KUKA KRL program: EPS_2_251806_MH07A_A_20260223023033.src

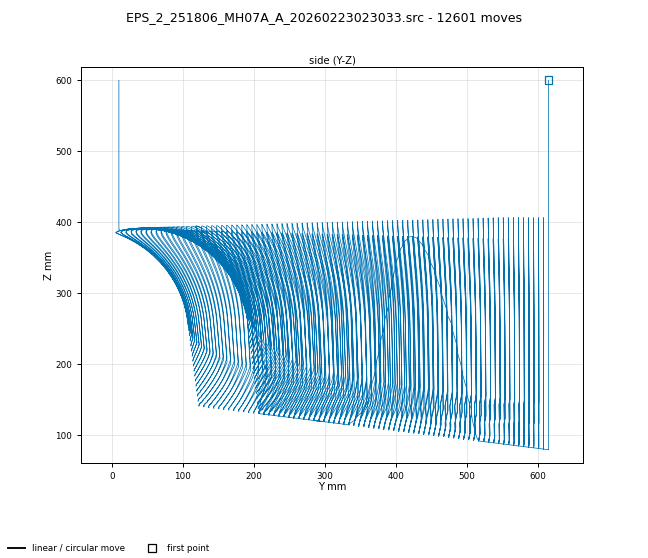
[picture p0: tool path of EPS_2_251806_MH07A_A_20260223023033.src, 12601 of 12603 moves have a stored position in this frame; points joined in program order, loops and branches not executed]
&ACCESS RVP
&REL 4
&COMMENT QRS 19112012
&PARAM EDITMASK = *
DEF PART()
EXT BAS (BAS_COMMAND :IN,REAL :IN )
INT I
BAS (#INITMOV,0 )

;KUKA QRS Post kuka4.cps  Date:22-06-2017 !

File_ID=3075

QRS_PRE_INIT()

;Init var - Until changes are made in qrs_pre_init
Outlet_Square_prg=0
Inlet_1_Square_prg=0
Inlet_2_Square_prg=0
Inlet_3_Square_prg=0
Inlet_4_Square_prg=0
Inlet_5_Square_prg=0

Outlet_1={X 0.000, Y 543.810, Z 281.000, B 0.000, E1 0.000 }
Inlet_1={X 0.000, Y 545.970, Z 251.000, B 0.000, E1 164.000 }
Outlet_1_type=251
Inlet_1_type=251
;QRS#1=Sidecore dimensions
;QRS#2=250-10" PVC SDR 35
;QRS#3=250-10" PVC SDR 35
;QRS#4=
;QRS#5=
;QRS#6=
;QRS#7=
;QRS#8=
;QRS#9=14M PSX
;QRS#10=14M PSX
;QRS#11=
;QRS#12=
;QRS#13=
;QRS#14=
;QRS#15=
;QRS#16=1220x127x686 2,25'
;QRS#17=EPS Height
;QRS#18=406,5
;QRS#19=*
;QRS#20= UPDATED VERSION 22-06-2017
;QRS#21=*
Outlet_Square=0100
Inlet_1_Square=0100
Inlet_2_Square=0
Inlet_3_Square=0
Inlet_4_Square=0
Inlet_5_Square=0
Mill_Square=1
Outlet_Square_Prg=205
Inlet_1_Square_prg=205

QRS_INIT()

$ADVANCE=5

; T1
PTP {E1 173.638,E2 173.638}
PTP {X 0,Y 615.462,A -85,B 0,C 180,E1 173.638,E2 173.638,E3 0,E4 0,E5 0,E6 0}
QRS_SPEED_INIT()
LIN {X 0,Y 615.462,Z 600,A -85,B 0,C 180,E1 173.638,E2 173.638,E3 0,E4 0,E5 0,E6 0} C_VEL
LIN {X 0,Y 615.462,Z 89.499,A -85,B 0,C 180,E1 173.638,E2 173.638} C_VEL
LIN {X 0,Y 615.462,Z 81.318,A -85,B 0,C 180,E1 173.638,E2 173.638} C_VEL
LIN {X 0,Y 615.456,Z 79.318,A -85,B 0,C 180,E1 173.452,E2 173.452} C_VEL
LIN {X 0,Y 615.494,Z 79.31,A -85,B 0,C 180,E1 170.804,E2 170.804} C_VEL
LIN {X 0,Y 615.478,Z 79.324,A -85,B 0,C 180,E1 168.142,E2 168.142} C_VEL
LIN {X 0,Y 615.453,Z 79.316,A -85,B 0,C 180,E1 165.453,E2 165.453} C_VEL
LIN {X 0,Y 615.495,Z 79.319,A -85,B 0,C 180,E1 162.733,E2 162.733} C_VEL
LIN {X 0,Y 615.448,Z 79.32,A -85,B 0,C 180,E1 159.969,E2 159.969} C_VEL
LIN {X 0,Y 615.45,Z 79.317,A -85,B 0,C 180,E1 157.664,E2 157.664} C_VEL
LIN {X 0,Y 615.497,Z 79.319,A -85,B 0,C 180,E1 155.012,E2 155.012} C_VEL
LIN {X 0,Y 615.485,Z 79.326,A -85,B 0,C 180,E1 152.826,E2 152.826} C_VEL
LIN {X 0,Y 615.437,Z 79.321,A -85,B 0,C 180,E1 150.215,E2 150.215} C_VEL
LIN {X 0,Y 615.461,Z 79.318,A -85,B 0,C 180,E1 147.674,E2 147.674} C_VEL
LIN {X 0,Y 615.498,Z 79.325,A -85,B 0,C 180,E1 145.19,E2 145.19} C_VEL
LIN {X 0,Y 615.444,Z 79.323,A -85,B 0,C 180,E1 142.759,E2 142.759} C_VEL
LIN {X 0,Y 615.46,Z 79.319,A -85,B 0,C 180,E1 139.915,E2 139.915} C_VEL
LIN {X 0,Y 615.5,Z 79.319,A -85,B 0,C 180,E1 137.653,E2 137.653} C_VEL
LIN {X 0,Y 615.431,Z 79.323,A -85,B 0,C 180,E1 134.931,E2 134.931} C_VEL
LIN {X 0,Y 615.465,Z 79.321,A -85,B 0,C 180,E1 132.083,E2 132.083} C_VEL
LIN {X 0,Y 615.489,Z 79.326,A -85,B 0,C 180,E1 129.751,E2 129.751} C_VEL
LIN {X 0,Y 615.429,Z 79.324,A -85,B 0,C 180,E1 127.247,E2 127.247} C_VEL
LIN {X 0,Y 615.431,Z 79.462,A -85,B 0,C 180,E1 126.587,E2 126.587} C_VEL
LIN {X 0,Y 615.47,Z 98.899,A -85,B 0,C 180,E1 123.78,E2 123.78} C_VEL
LIN {X 0,Y 615.473,Z 114.632,A -85,B 0,C 180,E1 121.538,E2 121.538} C_VEL
LIN {X 0,Y 615.488,Z 251.915,A -85,B 0,C 180,E1 119.892,E2 119.892} C_VEL
LIN {X 0,Y 615.49,Z 265.372,A -85,B 0,C 180,E1 119.604,E2 119.604} C_VEL
LIN {X 0,Y 615.481,Z 279.244,A -85,B 0,C 180,E1 119.173,E2 119.173} C_VEL
LIN {X 0,Y 615.488,Z 292.745,A -85,B 0,C 180,E1 118.609,E2 118.609} C_VEL
LIN {X 0,Y 615.495,Z 305.732,A -85,B 0,C 180,E1 117.916,E2 117.916} C_VEL
LIN {X 0,Y 615.497,Z 316.928,A -85,B 0,C 180,E1 117.178,E2 117.178} C_VEL
LIN {X 0,Y 615.497,Z 328.369,A -85,B 0,C 180,E1 116.262,E2 116.262} C_VEL
LIN {X 0,Y 615.494,Z 338.407,A -85,B 0,C 180,E1 115.286,E2 115.286} C_VEL
LIN {X 0,Y 615.497,Z 347.013,A -85,B 0,C 180,E1 114.272,E2 114.272} C_VEL
LIN {X 0,Y 615.496,Z 354.545,A -85,B 0,C 180,E1 113.2,E2 113.2} C_VEL
LIN {X 0,Y 615.498,Z 360.676,A -85,B 0,C 180,E1 112.137,E2 112.137} C_VEL
LIN {X 0,Y 615.498,Z 365.573,A -85,B 0,C 180,E1 111.081,E2 111.081} C_VEL
LIN {X 0,Y 615.489,Z 370.526,A -85,B 0,C 180,E1 109.686,E2 109.686} C_VEL
LIN {X 0,Y 615.497,Z 373.149,A -85,B 0,C 180,E1 108.62,E2 108.62} C_VEL
LIN {X 0,Y 615.493,Z 375.219,A -85,B 0,C 180,E1 107.271,E2 107.271} C_VEL
LIN {X 0,Y 615.493,Z 375.883,A -85,B 0,C 180,E1 105.906,E2 105.906} C_VEL
LIN {X 0,Y 615.497,Z 375.112,A -85,B 0,C 180,E1 104.55,E2 104.55} C_VEL
LIN {X 0,Y 615.495,Z 372.958,A -85,B 0,C 180,E1 103.202,E2 103.202} C_VEL
LIN {X 0,Y 615.49,Z 369.374,A -85,B 0,C 180,E1 101.862,E2 101.862} C_VEL
LIN {X 0,Y 615.495,Z 364.281,A -85,B 0,C 180,E1 100.528,E2 100.528} C_VEL
LIN {X 0,Y 615.495,Z 359.354,A -85,B 0,C 180,E1 99.531,E2 99.531} C_VEL
LIN {X 0,Y 615.495,Z 352.301,A -85,B 0,C 180,E1 98.372,E2 98.372} C_VEL
LIN {X 0,Y 615.495,Z 343.605,A -85,B 0,C 180,E1 97.216,E2 97.216} C_VEL
LIN {X 0,Y 615.497,Z 334.553,A -85,B 0,C 180,E1 96.228,E2 96.228} C_VEL
LIN {X 0,Y 615.497,Z 325.562,A -85,B 0,C 180,E1 95.406,E2 95.406} C_VEL
LIN {X 0,Y 615.498,Z 314.887,A -85,B 0,C 180,E1 94.585,E2 94.585} C_VEL
LIN {X 0,Y 615.485,Z 303.261,A -85,B 0,C 180,E1 93.847,E2 93.847} C_VEL
LIN {X 0,Y 615.495,Z 290.463,A -85,B 0,C 180,E1 93.192,E2 93.192} C_VEL
LIN {X 0,Y 615.496,Z 277.102,A -85,B 0,C 180,E1 92.66,E2 92.66} C_VEL
LIN {X 0,Y 615.47,Z 263.184,A -85,B 0,C 180,E1 92.25,E2 92.25} C_VEL
LIN {X 0,Y 615.451,Z 249.843,A -85,B 0,C 180,E1 91.985,E2 91.985} C_VEL
LIN {X 0,Y 615.447,Z 114.619,A -85,B 0,C 180,E1 90.369,E2 90.369} C_VEL
LIN {X 0,Y 615.485,Z 95.966,A -85,B 0,C 180,E1 87.71,E2 87.71} C_VEL
LIN {X 0,Y 615.485,Z 79.31,A -85,B 0,C 180,E1 85.293,E2 85.293} C_VEL
LIN {X 0,Y 615.473,Z 79.313,A -85,B 0,C 180,E1 82.785,E2 82.785} C_VEL
LIN {X 0,Y 615.499,Z 79.325,A -85,B 0,C 180,E1 80.139,E2 80.139} C_VEL
LIN {X 0,Y 615.491,Z 79.308,A -85,B 0,C 180,E1 77.471,E2 77.471} C_VEL
LIN {X 0,Y 615.472,Z 79.317,A -85,B 0,C 180,E1 74.775,E2 74.775} C_VEL
LIN {X 0,Y 615.483,Z 79.317,A -85,B 0,C 180,E1 72.044,E2 72.044} C_VEL
LIN {X 0,Y 615.479,Z 79.311,A -85,B 0,C 180,E1 69.27,E2 69.27} C_VEL
LIN {X 0,Y 615.486,Z 79.323,A -85,B 0,C 180,E1 66.445,E2 66.445} C_VEL
LIN {X 0,Y 615.485,Z 79.309,A -85,B 0,C 180,E1 63.557,E2 63.557} C_VEL
LIN {X 0,Y 615.476,Z 79.314,A -85,B 0,C 180,E1 61.343,E2 61.343} C_VEL
LIN {X 0,Y 615.488,Z 79.324,A -85,B 0,C 180,E1 58.906,E2 58.906} C_VEL
LIN {X 0,Y 615.496,Z 79.306,A -85,B 0,C 180,E1 55.98,E2 55.98} C_VEL
LIN {X 0,Y 615.49,Z 79.325,A -85,B 0,C 180,E1 53.057,E2 53.057} C_VEL
LIN {X 0,Y 615.487,Z 79.309,A -85,B 0,C 180,E1 50.251,E2 50.251} C_VEL
LIN {X 0,Y 615.478,Z 79.316,A -85,B 0,C 180,E1 47.648,E2 47.648} C_VEL
LIN {X 0,Y 615.481,Z 79.319,A -85,B 0,C 180,E1 44.933,E2 44.933} C_VEL
LIN {X 0,Y 615.481,Z 79.311,A -85,B 0,C 180,E1 42.081,E2 42.081} C_VEL
LIN {X 0,Y 615.481,Z 79.318,A -85,B 0,C 180,E1 39.746,E2 39.746} C_VEL
LIN {X 0,Y 615.477,Z 79.314,A -85,B 0,C 180,E1 36.937,E2 36.937} C_VEL
LIN {X 0,Y 615.487,Z 79.308,A -85,B 0,C 180,E1 34.703,E2 34.703} C_VEL
LIN {X 0,Y 615.481,Z 79.312,A -85,B 0,C 180,E1 32.332,E2 32.332} C_VEL
LIN {X 0,Y 615.493,Z 79.324,A -85,B 0,C 180,E1 29.798,E2 29.798} C_VEL
LIN {X 0,Y 615.476,Z 79.312,A -85,B 0,C 180,E1 27.046,E2 27.046} C_VEL
LIN {X 0,Y 615.482,Z 79.317,A -85,B 0,C 180,E1 24.269,E2 24.269} C_VEL
LIN {X 0,Y 615.475,Z 79.315,A -85,B 0,C 180,E1 21.429,E2 21.429} C_VEL
LIN {X 0,Y 615.482,Z 79.313,A -85,B 0,C 180,E1 18.607,E2 18.607} C_VEL
LIN {X 0,Y 615.481,Z 79.321,A -85,B 0,C 180,E1 15.903,E2 15.903} C_VEL
LIN {X 0,Y 615.491,Z 79.307,A -85,B 0,C 180,E1 13.198,E2 13.198} C_VEL
LIN {X 0,Y 615.488,Z 79.321,A -85,B 0,C 180,E1 10.524,E2 10.524} C_VEL
LIN {X 0,Y 615.472,Z 79.316,A -85,B 0,C 180,E1 7.873,E2 7.873} C_VEL
LIN {X 0,Y 615.492,Z 79.308,A -85,B 0,C 180,E1 5.239,E2 5.239} C_VEL
LIN {X 0,Y 615.495,Z 79.324,A -85,B 0,C 180,E1 2.616,E2 2.616} C_VEL
LIN {X 0,Y 615.472,Z 79.314,A -85,B 0,C 180,E1 -0.002,E2 -0.002} C_VEL
LIN {X 0,Y 615.489,Z 79.31,A -85,B 0,C 180,E1 -2.62,E2 -2.62} C_VEL
LIN {X 0,Y 615.49,Z 79.325,A -85,B 0,C 180,E1 -5.243,E2 -5.243} C_VEL
LIN {X 0,Y 615.47,Z 79.313,A -85,B 0,C 180,E1 -7.878,E2 -7.878} C_VEL
LIN {X 0,Y 615.486,Z 79.313,A -85,B 0,C 180,E1 -10.529,E2 -10.529} C_VEL
LIN {X 0,Y 615.475,Z 79.322,A -85,B 0,C 180,E1 -13.203,E2 -13.203} C_VEL
LIN {X 0,Y 615.486,Z 79.308,A -85,B 0,C 180,E1 -15.907,E2 -15.907} C_VEL
LIN {X 0,Y 615.487,Z 79.323,A -85,B 0,C 180,E1 -18.648,E2 -18.648} C_VEL
LIN {X 0,Y 615.469,Z 79.313,A -85,B 0,C 180,E1 -21.434,E2 -21.434} C_VEL
LIN {X 0,Y 615.487,Z 79.317,A -85,B 0,C 180,E1 -24.273,E2 -24.273} C_VEL
LIN {X 0,Y 615.466,Z 79.317,A -85,B 0,C 180,E1 -27.044,E2 -27.044} C_VEL
LIN {X 0,Y 615.492,Z 79.31,A -85,B 0,C 180,E1 -29.798,E2 -29.798} C_VEL
LIN {X 0,Y 615.489,Z 79.323,A -85,B 0,C 180,E1 -32.459,E2 -32.459} C_VEL
LIN {X 0,Y 615.464,Z 79.317,A -85,B 0,C 180,E1 -34.818,E2 -34.818} C_VEL
LIN {X 0,Y 615.48,Z 79.31,A -85,B 0,C 180,E1 -37.244,E2 -37.244} C_VEL
LIN {X 0,Y 615.496,Z 79.325,A -85,B 0,C 180,E1 -40.092,E2 -40.092} C_VEL
LIN {X 0,Y 615.473,Z 79.321,A -85,B 0,C 180,E1 -42.355,E2 -42.355} C_VEL
LIN {X 0,Y 615.476,Z 79.311,A -85,B 0,C 180,E1 -45.071,E2 -45.071} C_VEL
LIN {X 0,Y 615.494,Z 79.324,A -85,B 0,C 180,E1 -47.92,E2 -47.92} C_VEL
LIN {X 0,Y 615.465,Z 79.319,A -85,B 0,C 180,E1 -50.25,E2 -50.25} C_VEL
LIN {X 0,Y 615.49,Z 79.31,A -85,B 0,C 180,E1 -53.064,E2 -53.064} C_VEL
LIN {X 0,Y 615.469,Z 79.32,A -85,B 0,C 180,E1 -55.978,E2 -55.978} C_VEL
LIN {X 0,Y 615.461,Z 79.315,A -85,B 0,C 180,E1 -58.314,E2 -58.314} C_VEL
LIN {X 0,Y 615.476,Z 79.311,A -85,B 0,C 180,E1 -60.594,E2 -60.594} C_VEL
LIN {X 0,Y 615.478,Z 79.323,A -85,B 0,C 180,E1 -63.557,E2 -63.557} C_VEL
LIN {X 0,Y 615.459,Z 79.316,A -85,B 0,C 180,E1 -65.998,E2 -65.998} C_VEL
LIN {X 0,Y 615.485,Z 79.376,A -85,B 0,C 180,E1 -66.512,E2 -66.512} C_VEL
LIN {X 0,Y 615.489,Z 102.854,A -85,B 0,C 180,E1 -69.444,E2 -69.444} C_VEL
LIN {X 0,Y 615.492,Z 125.455,A -85,B 0,C 180,E1 -72.216,E2 -72.216} C_VEL
LIN {X 0,Y 615.493,Z 143.435,A -85,B 0,C 180,E1 -74.393,E2 -74.393} C_VEL
LIN {X 0,Y 615.477,Z 281.352,A -85,B 0,C 180,E1 -76.053,E2 -76.053} C_VEL
LIN {X 0,Y 615.489,Z 294.895,A -85,B 0,C 180,E1 -76.337,E2 -76.337} C_VEL
LIN {X 0,Y 615.488,Z 308.595,A -85,B 0,C 180,E1 -76.758,E2 -76.758} C_VEL
LIN {X 0,Y 615.494,Z 321.858,A -85,B 0,C 180,E1 -77.303,E2 -77.303} C_VEL
LIN {X 0,Y 615.483,Z 334.618,A -85,B 0,C 180,E1 -77.973,E2 -77.973} C_VEL
LIN {X 0,Y 615.499,Z 347.354,A -85,B 0,C 180,E1 -78.808,E2 -78.808} C_VEL
LIN {X 0,Y 615.498,Z 357.76,A -85,B 0,C 180,E1 -79.641,E2 -79.641} C_VEL
LIN {X 0,Y 615.496,Z 368.098,A -85,B 0,C 180,E1 -80.637,E2 -80.637} C_VEL
LIN {X 0,Y 615.497,Z 376.61,A -85,B 0,C 180,E1 -81.63,E2 -81.63} C_VEL
LIN {X 0,Y 615.496,Z 384.733,A -85,B 0,C 180,E1 -82.785,E2 -82.785} C_VEL
LIN {X 0,Y 615.497,Z 390.435,A -85,B 0,C 180,E1 -83.774,E2 -83.774} C_VEL
LIN {X 0,Y 615.495,Z 395.084,A -85,B 0,C 180,E1 -84.76,E2 -84.76} C_VEL
LIN {X 0,Y 615.496,Z 399.904,A -85,B 0,C 180,E1 -86.073,E2 -86.073} C_VEL
LIN {X 0,Y 615.495,Z 403.254,A -85,B 0,C 180,E1 -87.383,E2 -87.383} C_VEL
LIN {X 0,Y 615.49,Z 405.23,A -85,B 0,C 180,E1 -88.692,E2 -88.692} C_VEL
LIN {X 0,Y 615.493,Z 405.889,A -85,B 0,C 180,E1 -90.001,E2 -90.001} C_VEL
LIN {X 0,Y 615.49,Z 405.227,A -85,B 0,C 180,E1 -91.31,E2 -91.31} C_VEL
LIN {X 0,Y 615.495,Z 403.25,A -85,B 0,C 180,E1 -92.619,E2 -92.619} C_VEL
LIN {X 0,Y 615.496,Z 399.898,A -85,B 0,C 180,E1 -93.929,E2 -93.929} C_VEL
LIN {X 0,Y 615.495,Z 395.076,A -85,B 0,C 180,E1 -95.242,E2 -95.242} C_VEL
LIN {X 0,Y 615.495,Z 388.623,A -85,B 0,C 180,E1 -96.557,E2 -96.557} C_VEL
LIN {X 0,Y 615.498,Z 381.434,A -85,B 0,C 180,E1 -97.711,E2 -97.711} C_VEL
LIN {X 0,Y 615.497,Z 373.896,A -85,B 0,C 180,E1 -98.703,E2 -98.703} C_VEL
LIN {X 0,Y 615.496,Z 364.844,A -85,B 0,C 180,E1 -99.697,E2 -99.697} C_VEL
LIN {X 0,Y 615.497,Z 354.751,A -85,B 0,C 180,E1 -100.619,E2 -100.619} C_VEL
LIN {X 0,Y 615.498,Z 343.844,A -85,B 0,C 180,E1 -101.444,E2 -101.444} C_VEL
LIN {X 0,Y 615.484,Z 331.689,A -85,B 0,C 180,E1 -102.196,E2 -102.196} C_VEL
LIN {X 0,Y 615.486,Z 318.07,A -85,B 0,C 180,E1 -102.866,E2 -102.866} C_VEL
LIN {X 0,Y 615.488,Z 304.807,A -85,B 0,C 180,E1 -103.37,E2 -103.37} C_VEL
LIN {X 0,Y 615.487,Z 291.247,A -85,B 0,C 180,E1 -103.749,E2 -103.749} C_VEL
LIN {X 0,Y 615.478,Z 277.197,A -85,B 0,C 180,E1 -104.007,E2 -104.007} C_VEL
LIN {X 0,Y 615.493,Z 143.419,A -85,B 0,C 180,E1 -105.608,E2 -105.608} C_VEL
LIN {X 0,Y 615.483,Z 121.406,A -85,B 0,C 180,E1 -108.278,E2 -108.278} C_VEL
LIN {X 0,Y 615.475,Z 100.026,A -85,B 0,C 180,E1 -110.907,E2 -110.907} C_VEL
LIN {X 0,Y 615.483,Z 79.31,A -85,B 0,C 180,E1 -113.513,E2 -113.513} C_VEL
LIN {X 0,Y 615.466,Z 79.313,A -85,B 0,C 180,E1 -115.718,E2 -115.718} C_VEL
LIN {X 0,Y 615.49,Z 79.325,A -85,B 0,C 180,E1 -118.45,E2 -118.45} C_VEL
LIN {X 0,Y 615.487,Z 79.311,A -85,B 0,C 180,E1 -121.085,E2 -121.085} C_VEL
LIN {X 0,Y 615.468,Z 79.314,A -85,B 0,C 180,E1 -123.531,E2 -123.531} C_VEL
LIN {X 0,Y 615.471,Z 79.319,A -85,B 0,C 180,E1 -125.831,E2 -125.831} C_VEL
LIN {X 0,Y 615.492,Z 79.324,A -85,B 0,C 180,E1 -128.069,E2 -128.069} C_VEL
LIN {X 0,Y 615.482,Z 79.313,A -85,B 0,C 180,E1 -130.608,E2 -130.608} C_VEL
LIN {X 0,Y 615.471,Z 79.314,A -85,B 0,C 180,E1 -133.247,E2 -133.247} C_VEL
LIN {X 0,Y 615.49,Z 79.322,A -85,B 0,C 180,E1 -136.003,E2 -136.003} C_VEL
LIN {X 0,Y 615.481,Z 79.31,A -85,B 0,C 180,E1 -138.907,E2 -138.907} C_VEL
LIN {X 0,Y 615.475,Z 79.315,A -85,B 0,C 180,E1 -141.094,E2 -141.094} C_VEL
LIN {X 0,Y 615.484,Z 79.328,A -85,B 0,C 180,E1 -143.574,E2 -143.574} C_VEL
LIN {X 0,Y 615.494,Z 79.307,A -85,B 0,C 180,E1 -146.466,E2 -146.466} C_VEL
LIN {X 0,Y 615.484,Z 79.32,A -85,B 0,C 180,E1 -149.079,E2 -149.079} C_VEL
LIN {X 0,Y 615.477,Z 79.32,A -85,B 0,C 180,E1 -151.553,E2 -151.553} C_VEL
LIN {X 0,Y 615.486,Z 79.31,A -85,B 0,C 180,E1 -154.433,E2 -154.433} C_VEL
LIN {X 0,Y 615.484,Z 79.324,A -85,B 0,C 180,E1 -157.154,E2 -157.154} C_VEL
LIN {X 0,Y 615.484,Z 79.309,A -85,B 0,C 180,E1 -159.966,E2 -159.966} C_VEL
LIN {X 0,Y 615.491,Z 79.324,A -85,B 0,C 180,E1 -162.728,E2 -162.728} C_VEL
LIN {X 0,Y 615.471,Z 79.313,A -85,B 0,C 180,E1 -165.449,E2 -165.449} C_VEL
LIN {X 0,Y 615.486,Z 79.314,A -85,B 0,C 180,E1 -168.137,E2 -168.137} C_VEL
LIN {X 0,Y 615.475,Z 79.321,A -85,B 0,C 180,E1 -170.799,E2 -170.799} C_VEL
LIN {X 0,Y 615.478,Z 79.31,A -85,B 0,C 180,E1 -173.441,E2 -173.441} C_VEL
LIN {X 0,Y 615.491,Z 79.319,A -85,B 0,C 180,E1 -176.07,E2 -176.07} C_VEL
LIN {X 0,Y 615.462,Z 79.319,A -85,B 0,C 180,E1 -178.689,E2 -178.689} C_VEL
LIN {X 0,Y 615.484,Z 79.31,A -85,B 0,C 180,E1 -181.306,E2 -181.306} C_VEL
LIN {X 0,Y 615.49,Z 79.325,A -85,B 0,C 180,E1 -183.926,E2 -183.926} C_VEL
LIN {X 0,Y 615.456,Z 79.318,A -85,B 0,C 180,E1 -186.548,E2 -186.548} C_VEL
LIN {X 0,Y 614.803,Z 79.46,A -85,B 0,C 180,E1 -187.094,E2 -187.094} C_VEL
LIN {X 0,Y 611.99,Z 79.88,A -85,B 0,C 180,E1 -187.98,E2 -187.98} C_VEL
LIN {X 0,Y 609.6,Z 80.187,A -85,B 0,C 180,E1 -188.693,E2 -188.693} C_VEL
LIN {X 0,Y 608.559,Z 80.304,A -85,B 0,C 180,E1 -189.242,E2 -189.242} C_VEL
LIN {X 0,Y 608.466,Z 80.314,A -85,B 0,C 180,E1 -189.428,E2 -189.428} C_VEL
LIN {X 0,Y 608.45,Z 80.318,A -85,B 0,C 180,E1 -191.997,E2 -191.997} C_VEL
LIN {X 0,Y 608.427,Z 80.316,A -85,B 0,C 180,E1 -194.719,E2 -194.719} C_VEL
LIN {X 0,Y 608.449,Z 80.324,A -85,B 0,C 180,E1 -197.474,E2 -197.474} C_VEL
LIN {X 0,Y 608.432,Z 80.315,A -85,B 0,C 180,E1 -200.272,E2 -200.272} C_VEL
LIN {X 0,Y 608.454,Z 80.313,A -85,B 0,C 180,E1 -202.473,E2 -202.473} C_VEL
LIN {X 0,Y 608.44,Z 80.323,A -85,B 0,C 180,E1 -205.298,E2 -205.298} C_VEL
LIN {X 0,Y 608.43,Z 80.319,A -85,B 0,C 180,E1 -207.515,E2 -207.515} C_VEL
LIN {X 0,Y 608.425,Z 80.316,A -85,B 0,C 180,E1 -209.963,E2 -209.963} C_VEL
LIN {X 0,Y 608.438,Z 80.325,A -85,B 0,C 180,E1 -212.877,E2 -212.877} C_VEL
LIN {X 0,Y 608.417,Z 80.32,A -85,B 0,C 180,E1 -215.275,E2 -215.275} C_VEL
LIN {X 0,Y 608.434,Z 80.315,A -85,B 0,C 180,E1 -217.745,E2 -217.745} C_VEL
LIN {X 0,Y 608.437,Z 80.321,A -85,B 0,C 180,E1 -220.326,E2 -220.326} C_VEL
LIN {X 0,Y 608.413,Z 80.321,A -85,B 0,C 180,E1 -222.958,E2 -222.958} C_VEL
LIN {X 0,Y 608.406,Z 80.319,A -85,B 0,C 180,E1 -225.198,E2 -225.198} C_VEL
LIN {X 0,Y 608.443,Z 80.318,A -85,B 0,C 180,E1 -227.936,E2 -227.936} C_VEL
LIN {X 0,Y 608.408,Z 80.321,A -85,B 0,C 180,E1 -230.704,E2 -230.704} C_VEL
LIN {X 0,Y 608.433,Z 80.492,A -85,B 0,C 180,E1 -233.315,E2 -233.315} C_VEL
LIN {X 0,Y 608.523,Z 97.032,A -85,B 0,C 180,E1 -235.733,E2 -235.733} C_VEL
LIN {X 0,Y 608.499,Z 114.821,A -85,B 0,C 180,E1 -238.284,E2 -238.284} C_VEL
LIN {X 0,Y 608.618,Z 251.368,A -85,B 0,C 180,E1 -239.938,E2 -239.938} C_VEL
LIN {X 0,Y 608.587,Z 265.808,A -85,B 0,C 180,E1 -240.25,E2 -240.25} C_VEL
LIN {X 0,Y 608.552,Z 279.945,A -85,B 0,C 180,E1 -240.699,E2 -240.699} C_VEL
LIN {X 0,Y 608.556,Z 293.706,A -85,B 0,C 180,E1 -241.289,E2 -241.289} C_VEL
LIN {X 0,Y 608.537,Z 305.463,A -85,B 0,C 180,E1 -241.924,E2 -241.924} C_VEL
LIN {X 0,Y 608.524,Z 316.772,A -85,B 0,C 180,E1 -242.671,E2 -242.671} C_VEL
LIN {X 0,Y 608.494,Z 328.312,A -85,B 0,C 180,E1 -243.597,E2 -243.597} C_VEL
LIN {X 0,Y 608.47,Z 338.13,A -85,B 0,C 180,E1 -244.55,E2 -244.55} C_VEL
LIN {X 0,Y 608.472,Z 347.642,A -85,B 0,C 180,E1 -245.673,E2 -245.673} C_VEL
LIN {X 0,Y 608.452,Z 354.806,A -85,B 0,C 180,E1 -246.695,E2 -246.695} C_VEL
LIN {X 0,Y 608.452,Z 361.907,A -85,B 0,C 180,E1 -247.95,E2 -247.95} C_VEL
LIN {X 0,Y 608.442,Z 366.736,A -85,B 0,C 180,E1 -249.017,E2 -249.017} C_VEL
LIN {X 0,Y 608.43,Z 370.458,A -85,B 0,C 180,E1 -250.076,E2 -250.076} C_VEL
LIN {X 0,Y 608.423,Z 373.589,A -85,B 0,C 180,E1 -251.285,E2 -251.285} C_VEL
LIN {X 0,Y 608.414,Z 375.595,A -85,B 0,C 180,E1 -252.521,E2 -252.521} C_VEL
LIN {X 0,Y 608.429,Z 376.473,A -85,B 0,C 180,E1 -253.904,E2 -253.904} C_VEL
LIN {X 0,Y 608.42,Z 375.927,A -85,B 0,C 180,E1 -255.277,E2 -255.277} C_VEL
LIN {X 0,Y 608.436,Z 373.942,A -85,B 0,C 180,E1 -256.642,E2 -256.642} C_VEL
LIN {X 0,Y 608.432,Z 370.506,A -85,B 0,C 180,E1 -257.999,E2 -257.999} C_VEL
LIN {X 0,Y 608.434,Z 365.561,A -85,B 0,C 180,E1 -259.349,E2 -259.349} C_VEL
LIN {X 0,Y 608.463,Z 360.794,A -85,B 0,C 180,E1 -260.358,E2 -260.358} C_VEL
LIN {X 0,Y 608.458,Z 353.91,A -85,B 0,C 180,E1 -261.53,E2 -261.53} C_VEL
LIN {X 0,Y 608.463,Z 345.405,A -85,B 0,C 180,E1 -262.7,E2 -262.7} C_VEL
LIN {X 0,Y 608.48,Z 336.577,A -85,B 0,C 180,E1 -263.7,E2 -263.7} C_VEL
LIN {X 0,Y 608.497,Z 325.954,A -85,B 0,C 180,E1 -264.698,E2 -264.698} C_VEL
LIN {X 0,Y 608.516,Z 314.119,A -85,B 0,C 180,E1 -265.611,E2 -265.611} C_VEL
LIN {X 0,Y 608.528,Z 302.23,A -85,B 0,C 180,E1 -266.357,E2 -266.357} C_VEL
LIN {X 0,Y 608.548,Z 289.045,A -85,B 0,C 180,E1 -267.02,E2 -267.02} C_VEL
LIN {X 0,Y 608.578,Z 275.168,A -85,B 0,C 180,E1 -267.558,E2 -267.558} C_VEL
LIN {X 0,Y 608.584,Z 261.299,A -85,B 0,C 180,E1 -267.952,E2 -267.952} C_VEL
LIN {X 0,Y 608.564,Z 246.752,A -85,B 0,C 180,E1 -268.221,E2 -268.221} C_VEL
LIN {X 0,Y 608.487,Z 115.112,A -85,B 0,C 180,E1 -269.803,E2 -269.803} C_VEL
LIN {X 0,Y 608.452,Z 114.575,A -85,B 0,C 180,E1 -269.834,E2 -269.834} C_VEL
LIN {X 0,Y 608.542,Z 95.029,A -85,B 0,C 180,E1 -272.647,E2 -272.647} C_VEL
LIN {X 0,Y 608.457,Z 80.314,A -85,B 0,C 180,E1 -274.803,E2 -274.803} C_VEL
LIN {X 0,Y 608.462,Z 80.313,A -85,B 0,C 180,E1 -277.298,E2 -277.298} C_VEL
LIN {X 0,Y 608.463,Z 80.32,A -85,B 0,C 180,E1 -279.976,E2 -279.976} C_VEL
LIN {X 0,Y 608.473,Z 80.31,A -85,B 0,C 180,E1 -282.676,E2 -282.676} C_VEL
LIN {X 0,Y 608.458,Z 80.318,A -85,B 0,C 180,E1 -285.405,E2 -285.405} C_VEL
LIN {X 0,Y 608.442,Z 80.322,A -85,B 0,C 180,E1 -287.476,E2 -287.476} C_VEL
LIN {X 0,Y 608.458,Z 80.313,A -85,B 0,C 180,E1 -290.273,E2 -290.273} C_VEL
LIN {X 0,Y 608.462,Z 80.311,A -85,B 0,C 180,E1 -292.487,E2 -292.487} C_VEL
LIN {X 0,Y 608.445,Z 80.323,A -85,B 0,C 180,E1 -295.3,E2 -295.3} C_VEL
LIN {X 0,Y 608.442,Z 80.321,A -85,B 0,C 180,E1 -297.517,E2 -297.517} C_VEL
LIN {X 0,Y 608.485,Z 80.309,A -85,B 0,C 180,E1 -299.982,E2 -299.982} C_VEL
LIN {X 0,Y 608.448,Z 80.319,A -85,B 0,C 180,E1 -302.879,E2 -302.879} C_VEL
LIN {X 0,Y 608.464,Z 80.318,A -85,B 0,C 180,E1 -305.275,E2 -305.275} C_VEL
LIN {X 0,Y 608.464,Z 80.312,A -85,B 0,C 180,E1 -307.745,E2 -307.745} C_VEL
LIN {X 0,Y 608.448,Z 80.315,A -85,B 0,C 180,E1 -310.334,E2 -310.334} C_VEL
LIN {X 0,Y 608.447,Z 80.321,A -85,B 0,C 180,E1 -312.959,E2 -312.959} C_VEL
LIN {X 0,Y 608.455,Z 80.312,A -85,B 0,C 180,E1 -315.735,E2 -315.735} C_VEL
LIN {X 0,Y 608.458,Z 80.313,A -85,B 0,C 180,E1 -317.943,E2 -317.943} C_VEL
LIN {X 0,Y 608.461,Z 80.32,A -85,B 0,C 180,E1 -320.702,E2 -320.702} C_VEL
LIN {X 0,Y 608.448,Z 80.315,A -85,B 0,C 180,E1 -323.089,E2 -323.089} C_VEL
LIN {X 0,Y 608.466,Z 80.311,A -85,B 0,C 180,E1 -325.535,E2 -325.535} C_VEL
LIN {X 0,Y 608.461,Z 80.315,A -85,B 0,C 180,E1 -327.909,E2 -327.909} C_VEL
LIN {X 0,Y 608.476,Z 80.319,A -85,B 0,C 180,E1 -330.225,E2 -330.225} C_VEL
LIN {X 0,Y 608.465,Z 80.313,A -85,B 0,C 180,E1 -332.793,E2 -332.793} C_VEL
LIN {X 0,Y 608.448,Z 80.314,A -85,B 0,C 180,E1 -335.432,E2 -335.432} C_VEL
LIN {X 0,Y 608.461,Z 80.317,A -85,B 0,C 180,E1 -338.311,E2 -338.311} C_VEL
LIN {X 0,Y 608.445,Z 80.314,A -85,B 0,C 180,E1 -341.133,E2 -341.133} C_VEL
LIN {X 0,Y 608.456,Z 80.322,A -85,B 0,C 180,E1 -343.909,E2 -343.909} C_VEL
LIN {X 0,Y 608.464,Z 80.311,A -85,B 0,C 180,E1 -346.646,E2 -346.646} C_VEL
LIN {X 0,Y 608.464,Z 80.316,A -85,B 0,C 180,E1 -349.353,E2 -349.353} C_VEL
LIN {X 0,Y 608.466,Z 80.314,A -85,B 0,C 180,E1 -352.035,E2 -352.035} C_VEL
LIN {X 0,Y 608.469,Z 80.311,A -85,B 0,C 180,E1 -354.701,E2 -354.701} C_VEL
LIN {X 0,Y 608.484,Z 80.318,A -85,B 0,C 180,E1 -357.354,E2 -357.354} C_VEL
LIN {X 0,Y 608.463,Z 80.313,A -85,B 0,C 180,E1 -360.002,E2 -360.002} C_VEL
LIN {X 0,Y 608.479,Z 80.311,A -85,B 0,C 180,E1 -362.65,E2 -362.65} C_VEL
LIN {X 0,Y 608.467,Z 80.319,A -85,B 0,C 180,E1 -365.304,E2 -365.304} C_VEL
LIN {X 0,Y 608.465,Z 80.311,A -85,B 0,C 180,E1 -367.969,E2 -367.969} C_VEL
LIN {X 0,Y 608.465,Z 80.315,A -85,B 0,C 180,E1 -370.652,E2 -370.652} C_VEL
LIN {X 0,Y 608.454,Z 80.316,A -85,B 0,C 180,E1 -373.358,E2 -373.358} C_VEL
LIN {X 0,Y 608.46,Z 80.312,A -85,B 0,C 180,E1 -376.096,E2 -376.096} C_VEL
LIN {X 0,Y 608.45,Z 80.322,A -85,B 0,C 180,E1 -378.871,E2 -378.871} C_VEL
LIN {X 0,Y 608.46,Z 80.312,A -85,B 0,C 180,E1 -381.693,E2 -381.693} C_VEL
LIN {X 0,Y 608.447,Z 80.324,A -85,B 0,C 180,E1 -384.573,E2 -384.573} C_VEL
LIN {X 0,Y 608.462,Z 80.312,A -85,B 0,C 180,E1 -387.207,E2 -387.207} C_VEL
LIN {X 0,Y 608.47,Z 80.314,A -85,B 0,C 180,E1 -389.974,E2 -389.974} C_VEL
LIN {X 0,Y 608.452,Z 80.315,A -85,B 0,C 180,E1 -392.881,E2 -392.881} C_VEL
LIN {X 0,Y 608.439,Z 80.314,A -85,B 0,C 180,E1 -395.279,E2 -395.279} C_VEL
LIN {X 0,Y 608.47,Z 80.32,A -85,B 0,C 180,E1 -398.243,E2 -398.243} C_VEL
LIN {X 0,Y 608.462,Z 80.312,A -85,B 0,C 180,E1 -401.344,E2 -401.344} C_VEL
LIN {X 0,Y 608.452,Z 80.318,A -85,B 0,C 180,E1 -404.265,E2 -404.265} C_VEL
LIN {X 0,Y 608.444,Z 80.314,A -85,B 0,C 180,E1 -407.041,E2 -407.041} C_VEL
LIN {X 0,Y 608.454,Z 80.321,A -85,B 0,C 180,E1 -409.698,E2 -409.698} C_VEL
LIN {X 0,Y 608.46,Z 80.314,A -85,B 0,C 180,E1 -412.255,E2 -412.255} C_VEL
LIN {X 0,Y 608.453,Z 80.315,A -85,B 0,C 180,E1 -415.095,E2 -415.095} C_VEL
LIN {X 0,Y 608.46,Z 80.316,A -85,B 0,C 180,E1 -417.907,E2 -417.907} C_VEL
LIN {X 0,Y 608.446,Z 80.314,A -85,B 0,C 180,E1 -420.221,E2 -420.221} C_VEL
LIN {X 0,Y 608.481,Z 80.311,A -85,B 0,C 180,E1 -422.793,E2 -422.793} C_VEL
LIN {X 0,Y 608.445,Z 80.323,A -85,B 0,C 180,E1 -425.43,E2 -425.43} C_VEL
LIN {X 0,Y 608.477,Z 80.436,A -85,B 0,C 180,E1 -426.36,E2 -426.36} C_VEL
LIN {X 0,Y 608.596,Z 97.216,A -85,B 0,C 180,E1 -428.492,E2 -428.492} C_VEL
LIN {X 0,Y 608.532,Z 119.494,A -85,B 0,C 180,E1 -431.268,E2 -431.268} C_VEL
LIN {X 0,Y 608.521,Z 142.434,A -85,B 0,C 180,E1 -434.081,E2 -434.081} C_VEL
LIN {X 0,Y 608.514,Z 143.582,A -85,B 0,C 180,E1 -434.221,E2 -434.221} C_VEL
LIN {X 0,Y 608.598,Z 281.51,A -85,B 0,C 180,E1 -435.895,E2 -435.895} C_VEL
LIN {X 0,Y 608.603,Z 295.662,A -85,B 0,C 180,E1 -436.201,E2 -436.201} C_VEL
LIN {X 0,Y 608.579,Z 309.738,A -85,B 0,C 180,E1 -436.647,E2 -436.647} C_VEL
LIN {X 0,Y 608.554,Z 321.905,A -85,B 0,C 180,E1 -437.156,E2 -437.156} C_VEL
LIN {X 0,Y 608.511,Z 334.698,A -85,B 0,C 180,E1 -437.833,E2 -437.833} C_VEL
LIN {X 0,Y 608.499,Z 347.485,A -85,B 0,C 180,E1 -438.678,E2 -438.678} C_VEL
LIN {X 0,Y 608.495,Z 357.943,A -85,B 0,C 180,E1 -439.52,E2 -439.52} C_VEL
LIN {X 0,Y 608.479,Z 368.344,A -85,B 0,C 180,E1 -440.528,E2 -440.528} C_VEL
LIN {X 0,Y 608.464,Z 376.922,A -85,B 0,C 180,E1 -441.532,E2 -441.532} C_VEL
LIN {X 0,Y 608.461,Z 385.119,A -85,B 0,C 180,E1 -442.702,E2 -442.702} C_VEL
LIN {X 0,Y 608.444,Z 391.55,A -85,B 0,C 180,E1 -443.832,E2 -443.832} C_VEL
LIN {X 0,Y 608.435,Z 396.965,A -85,B 0,C 180,E1 -445.031,E2 -445.031} C_VEL
LIN {X 0,Y 608.434,Z 400.444,A -85,B 0,C 180,E1 -446.027,E2 -446.027} C_VEL
LIN {X 0,Y 608.423,Z 403.833,A -85,B 0,C 180,E1 -447.353,E2 -447.353} C_VEL
LIN {X 0,Y 608.442,Z 405.832,A -85,B 0,C 180,E1 -448.677,E2 -448.677} C_VEL
LIN {X 0,Y 608.433,Z 406.5,A -85,B 0,C 180,E1 -450.001,E2 -450.001} C_VEL
LIN {X 0,Y 608.442,Z 405.829,A -85,B 0,C 180,E1 -451.325,E2 -451.325} C_VEL
LIN {X 0,Y 608.423,Z 403.829,A -85,B 0,C 180,E1 -452.649,E2 -452.649} C_VEL
LIN {X 0,Y 608.434,Z 400.438,A -85,B 0,C 180,E1 -453.975,E2 -453.975} C_VEL
LIN {X 0,Y 608.439,Z 395.564,A -85,B 0,C 180,E1 -455.303,E2 -455.303} C_VEL
LIN {X 0,Y 608.447,Z 389.207,A -85,B 0,C 180,E1 -456.604,E2 -456.604} C_VEL
LIN {X 0,Y 608.454,Z 381.791,A -85,B 0,C 180,E1 -457.801,E2 -457.801} C_VEL
LIN {X 0,Y 608.473,Z 372.815,A -85,B 0,C 180,E1 -458.972,E2 -458.972} C_VEL
LIN {X 0,Y 608.473,Z 363.381,A -85,B 0,C 180,E1 -459.978,E2 -459.978} C_VEL
LIN {X 0,Y 608.506,Z 352.049,A -85,B 0,C 180,E1 -460.973,E2 -460.973} C_VEL
LIN {X 0,Y 608.531,Z 340.134,A -85,B 0,C 180,E1 -461.83,E2 -461.83} C_VEL
LIN {X 0,Y 608.53,Z 327.055,A -85,B 0,C 180,E1 -462.592,E2 -462.592} C_VEL
LIN {X 0,Y 608.55,Z 314.149,A -85,B 0,C 180,E1 -463.185,E2 -463.185} C_VEL
LIN {X 0,Y 608.59,Z 300.148,A -85,B 0,C 180,E1 -463.673,E2 -463.673} C_VEL
LIN {X 0,Y 608.602,Z 286.402,A -85,B 0,C 180,E1 -464.014,E2 -464.014} C_VEL
LIN {X 0,Y 608.591,Z 270.086,A -85,B 0,C 180,E1 -464.259,E2 -464.259} C_VEL
LIN {X 0,Y 608.53,Z 143.566,A -85,B 0,C 180,E1 -465.781,E2 -465.781} C_VEL
LIN {X 0,Y 608.537,Z 121.421,A -85,B 0,C 180,E1 -468.494,E2 -468.494} C_VEL
LIN {X 0,Y 608.561,Z 100.026,A -85,B 0,C 180,E1 -471.156,E2 -471.156} C_VEL
LIN {X 0,Y 608.57,Z 80.95,A -85,B 0,C 180,E1 -473.57,E2 -473.57} C_VEL
LIN {X 0,Y 608.447,Z 80.316,A -85,B 0,C 180,E1 -473.666,E2 -473.666} C_VEL
LIN {X 0,Y 608.434,Z 80.317,A -85,B 0,C 180,E1 -476.037,E2 -476.037} C_VEL
LIN {X 0,Y 608.477,Z 80.319,A -85,B 0,C 180,E1 -478.62,E2 -478.62} C_VEL
LIN {X 0,Y 608.449,Z 80.314,A -85,B 0,C 180,E1 -481.318,E2 -481.318} C_VEL
LIN {X 0,Y 608.454,Z 80.315,A -85,B 0,C 180,E1 -483.731,E2 -483.731} C_VEL
LIN {X 0,Y 608.45,Z 80.321,A -85,B 0,C 180,E1 -486.093,E2 -486.093} C_VEL
LIN {X 0,Y 608.477,Z 80.313,A -85,B 0,C 180,E1 -488.588,E2 -488.588} C_VEL
LIN {X 0,Y 608.453,Z 80.314,A -85,B 0,C 180,E1 -491.34,E2 -491.34} C_VEL
LIN {X 0,Y 608.458,Z 80.317,A -85,B 0,C 180,E1 -494.263,E2 -494.263} C_VEL
LIN {X 0,Y 608.449,Z 80.314,A -85,B 0,C 180,E1 -497.039,E2 -497.039} C_VEL
LIN {X 0,Y 608.464,Z 80.322,A -85,B 0,C 180,E1 -499.696,E2 -499.696} C_VEL
LIN {X 0,Y 608.468,Z 80.312,A -85,B 0,C 180,E1 -502.252,E2 -502.252} C_VEL
LIN {X 0,Y 608.447,Z 80.317,A -85,B 0,C 180,E1 -505.096,E2 -505.096} C_VEL
LIN {X 0,Y 608.464,Z 80.314,A -85,B 0,C 180,E1 -507.904,E2 -507.904} C_VEL
LIN {X 0,Y 608.474,Z 80.31,A -85,B 0,C 180,E1 -510.219,E2 -510.219} C_VEL
LIN {X 0,Y 608.478,Z 80.313,A -85,B 0,C 180,E1 -512.794,E2 -512.794} C_VEL
LIN {X 0,Y 608.45,Z 80.318,A -85,B 0,C 180,E1 -515.427,E2 -515.427} C_VEL
LIN {X 0,Y 608.466,Z 80.312,A -85,B 0,C 180,E1 -518.307,E2 -518.307} C_VEL
LIN {X 0,Y 608.467,Z 80.315,A -85,B 0,C 180,E1 -521.287,E2 -521.287} C_VEL
LIN {X 0,Y 608.459,Z 80.312,A -85,B 0,C 180,E1 -523.904,E2 -523.904} C_VEL
LIN {X 0,Y 608.466,Z 80.321,A -85,B 0,C 180,E1 -526.642,E2 -526.642} C_VEL
LIN {X 0,Y 608.452,Z 80.313,A -85,B 0,C 180,E1 -529.348,E2 -529.348} C_VEL
LIN {X 0,Y 608.478,Z 80.313,A -85,B 0,C 180,E1 -532.031,E2 -532.031} C_VEL
LIN {X 0,Y 608.451,Z 80.318,A -85,B 0,C 180,E1 -534.696,E2 -534.696} C_VEL
LIN {X 0,Y 608.473,Z 80.31,A -85,B 0,C 180,E1 -537.35,E2 -537.35} C_VEL
LIN {X 0,Y 608.484,Z 80.317,A -85,B 0,C 180,E1 -539.998,E2 -539.998} C_VEL
LIN {X 0,Y 608.455,Z 80.314,A -85,B 0,C 180,E1 -542.646,E2 -542.646} C_VEL
LIN {X 0,Y 608.468,Z 80.312,A -85,B 0,C 180,E1 -545.299,E2 -545.299} C_VEL
LIN {X 0,Y 608.474,Z 80.318,A -85,B 0,C 180,E1 -547.965,E2 -547.965} C_VEL
LIN {X 0,Y 608.466,Z 80.314,A -85,B 0,C 180,E1 -549.428,E2 -549.428} C_VEL
LIN {X 0,Y 607.779,Z 80.404,A -85,B 0,C 180,E1 -549.981,E2 -549.981} C_VEL
LIN {X 0,Y 604.92,Z 80.758,A -85,B 0,C 180,E1 -550.878,E2 -550.878} C_VEL
LIN {X 0,Y 602.516,Z 81.061,A -85,B 0,C 180,E1 -551.599,E2 -551.599} C_VEL
LIN {X 0,Y 601.482,Z 81.184,A -85,B 0,C 180,E1 -552.156,E2 -552.156} C_VEL
LIN {X 0,Y 601.397,Z 81.193,A -85,B 0,C 180,E1 -552.344,E2 -552.344} C_VEL
LIN {X 0,Y 601.4,Z 81.193,A -85,B 0,C 180,E1 -554.895,E2 -554.895} C_VEL
LIN {X 0,Y 601.408,Z 81.193,A -85,B 0,C 180,E1 -556.984,E2 -556.984} C_VEL
LIN {X 0,Y 601.39,Z 81.196,A -85,B 0,C 180,E1 -559.807,E2 -559.807} C_VEL
LIN {X 0,Y 601.407,Z 81.192,A -85,B 0,C 180,E1 -562.68,E2 -562.68} C_VEL
LIN {X 0,Y 601.39,Z 81.198,A -85,B 0,C 180,E1 -564.876,E2 -564.876} C_VEL
LIN {X 0,Y 601.407,Z 81.196,A -85,B 0,C 180,E1 -567.36,E2 -567.36} C_VEL
LIN {X 0,Y 601.391,Z 81.196,A -85,B 0,C 180,E1 -569.391,E2 -569.391} C_VEL
LIN {X 0,Y 601.38,Z 81.194,A -85,B 0,C 180,E1 -571.724,E2 -571.724} C_VEL
LIN {X 0,Y 601.403,Z 81.192,A -85,B 0,C 180,E1 -574.116,E2 -574.116} C_VEL
LIN {X 0,Y 601.386,Z 81.201,A -85,B 0,C 180,E1 -576.58,E2 -576.58} C_VEL
LIN {X 0,Y 601.375,Z 81.198,A -85,B 0,C 180,E1 -579.125,E2 -579.125} C_VEL
LIN {X 0,Y 601.395,Z 81.193,A -85,B 0,C 180,E1 -581.763,E2 -581.763} C_VEL
LIN {X 0,Y 601.404,Z 81.2,A -85,B 0,C 180,E1 -584.532,E2 -584.532} C_VEL
LIN {X 0,Y 601.352,Z 81.198,A -85,B 0,C 180,E1 -587.323,E2 -587.323} C_VEL
LIN {X 0,Y 601.378,Z 81.202,A -85,B 0,C 180,E1 -590.001,E2 -590.001} C_VEL
LIN {X 0,Y 601.402,Z 81.196,A -85,B 0,C 180,E1 -592.616,E2 -592.616} C_VEL
LIN {X 0,Y 601.38,Z 81.291,A -85,B 0,C 180,E1 -593.18,E2 -593.18} C_VEL
LIN {X 0,Y 601.532,Z 89.657,A -85,B 0,C 180,E1 -594.426,E2 -594.426} C_VEL
LIN {X 0,Y 601.493,Z 106.192,A -85,B 0,C 180,E1 -596.851,E2 -596.851} C_VEL
LIN {X 0,Y 601.473,Z 114.651,A -85,B 0,C 180,E1 -598.079,E2 -598.079} C_VEL
LIN {X 0,Y 601.815,Z 118.473,A -85,B 0,C 180,E1 -598.149,E2 -598.149} C_VEL
LIN {X 0,Y 601.735,Z 251.743,A -85,B 0,C 180,E1 -599.78,E2 -599.78} C_VEL
LIN {X 0,Y 601.693,Z 265.901,A -85,B 0,C 180,E1 -600.091,E2 -600.091} C_VEL
LIN {X 0,Y 601.647,Z 279.392,A -85,B 0,C 180,E1 -600.522,E2 -600.522} C_VEL
LIN {X 0,Y 601.598,Z 292.907,A -85,B 0,C 180,E1 -601.099,E2 -601.099} C_VEL
LIN {X 0,Y 601.573,Z 305.107,A -85,B 0,C 180,E1 -601.76,E2 -601.76} C_VEL
LIN {X 0,Y 601.524,Z 316.93,A -85,B 0,C 180,E1 -602.549,E2 -602.549} C_VEL
LIN {X 0,Y 601.456,Z 328.058,A -85,B 0,C 180,E1 -603.451,E2 -603.451} C_VEL
LIN {X 0,Y 601.417,Z 337.583,A -85,B 0,C 180,E1 -604.381,E2 -604.381} C_VEL
LIN {X 0,Y 601.415,Z 346.684,A -85,B 0,C 180,E1 -605.448,E2 -605.448} C_VEL
LIN {X 0,Y 601.393,Z 354.676,A -85,B 0,C 180,E1 -606.588,E2 -606.588} C_VEL
LIN {X 0,Y 601.365,Z 361.12,A -85,B 0,C 180,E1 -607.718,E2 -607.718} C_VEL
LIN {X 0,Y 601.374,Z 365.898,A -85,B 0,C 180,E1 -608.759,E2 -608.759} C_VEL
LIN {X 0,Y 601.332,Z 369.834,A -85,B 0,C 180,E1 -609.831,E2 -609.831} C_VEL
LIN {X 0,Y 601.334,Z 373.461,A -85,B 0,C 180,E1 -611.192,E2 -611.192} C_VEL
LIN {X 0,Y 601.307,Z 375.369,A -85,B 0,C 180,E1 -612.308,E2 -612.308} C_VEL
LIN {X 0,Y 601.343,Z 376.428,A -85,B 0,C 180,E1 -613.71,E2 -613.71} C_VEL
LIN {X 0,Y 601.311,Z 376.065,A -85,B 0,C 180,E1 -615.099,E2 -615.099} C_VEL
LIN {X 0,Y 601.361,Z 375.211,A -85,B 0,C 180,E1 -615.914,E2 -615.914} C_VEL
LIN {X 0,Y 601.325,Z 372.88,A -85,B 0,C 180,E1 -617.169,E2 -617.169} C_VEL
LIN {X 0,Y 601.348,Z 368.928,A -85,B 0,C 180,E1 -618.539,E2 -618.539} C_VEL
LIN {X 0,Y 601.347,Z 363.391,A -85,B 0,C 180,E1 -619.903,E2 -619.903} C_VEL
LIN {X 0,Y 601.383,Z 357.148,A -85,B 0,C 180,E1 -621.091,E2 -621.091} C_VEL
LIN {X 0,Y 601.382,Z 349.408,A -85,B 0,C 180,E1 -622.276,E2 -622.276} C_VEL
LIN {X 0,Y 601.44,Z 340.204,A -85,B 0,C 180,E1 -623.42,E2 -623.42} C_VEL
LIN {X 0,Y 601.455,Z 329.97,A -85,B 0,C 180,E1 -624.467,E2 -624.467} C_VEL
LIN {X 0,Y 601.497,Z 318.973,A -85,B 0,C 180,E1 -625.392,E2 -625.392} C_VEL
LIN {X 0,Y 601.532,Z 306.751,A -85,B 0,C 180,E1 -626.231,E2 -626.231} C_VEL
LIN {X 0,Y 601.588,Z 294.726,A -85,B 0,C 180,E1 -626.902,E2 -626.902} C_VEL
LIN {X 0,Y 601.638,Z 281.47,A -85,B 0,C 180,E1 -627.488,E2 -627.488} C_VEL
LIN {X 0,Y 601.683,Z 266.927,A -85,B 0,C 180,E1 -627.97,E2 -627.97} C_VEL
LIN {X 0,Y 601.682,Z 253.205,A -85,B 0,C 180,E1 -628.284,E2 -628.284} C_VEL
LIN {X 0,Y 601.713,Z 227.828,A -85,B 0,C 180,E1 -628.619,E2 -628.619} C_VEL
LIN {X 0,Y 601.749,Z 116.429,A -85,B 0,C 180,E1 -629.968,E2 -629.968} C_VEL
LIN {X 0,Y 601.438,Z 114.738,A -85,B 0,C 180,E1 -629.999,E2 -629.999} C_VEL
LIN {X 0,Y 601.556,Z 96.344,A -85,B 0,C 180,E1 -632.678,E2 -632.678} C_VEL
LIN {X 0,Y 601.501,Z 81.611,A -85,B 0,C 180,E1 -634.858,E2 -634.858} C_VEL
LIN {X 0,Y 601.43,Z 81.191,A -85,B 0,C 180,E1 -634.943,E2 -634.943} C_VEL
LIN {X 0,Y 601.428,Z 81.191,A -85,B 0,C 180,E1 -637.384,E2 -637.384} C_VEL
LIN {X 0,Y 601.436,Z 81.193,A -85,B 0,C 180,E1 -640.094,E2 -640.094} C_VEL
LIN {X 0,Y 601.441,Z 81.187,A -85,B 0,C 180,E1 -642.827,E2 -642.827} C_VEL
LIN {X 0,Y 601.411,Z 81.199,A -85,B 0,C 180,E1 -645.59,E2 -645.59} C_VEL
LIN {X 0,Y 601.39,Z 81.201,A -85,B 0,C 180,E1 -647.687,E2 -647.687} C_VEL
LIN {X 0,Y 601.421,Z 81.189,A -85,B 0,C 180,E1 -650.521,E2 -650.521} C_VEL
LIN {X 0,Y 601.409,Z 81.2,A -85,B 0,C 180,E1 -653.41,E2 -653.41} C_VEL
LIN {X 0,Y 601.395,Z 81.192,A -85,B 0,C 180,E1 -656.363,E2 -656.363} C_VEL
LIN {X 0,Y 601.424,Z 81.191,A -85,B 0,C 180,E1 -658.795,E2 -658.795} C_VEL
LIN {X 0,Y 601.416,Z 81.195,A -85,B 0,C 180,E1 -661.461,E2 -661.461} C_VEL
LIN {X 0,Y 601.415,Z 81.189,A -85,B 0,C 180,E1 -664.118,E2 -664.118} C_VEL
LIN {X 0,Y 601.4,Z 81.195,A -85,B 0,C 180,E1 -666.582,E2 -666.582} C_VEL
LIN {X 0,Y 601.429,Z 81.189,A -85,B 0,C 180,E1 -669.54,E2 -669.54} C_VEL
LIN {X 0,Y 601.415,Z 81.196,A -85,B 0,C 180,E1 -672.596,E2 -672.596} C_VEL
LIN {X 0,Y 601.426,Z 81.189,A -85,B 0,C 180,E1 -675.487,E2 -675.487} C_VEL
LIN {X 0,Y 601.414,Z 81.196,A -85,B 0,C 180,E1 -678.406,E2 -678.406} C_VEL
LIN {X 0,Y 601.42,Z 81.194,A -85,B 0,C 180,E1 -680.879,E2 -680.879} C_VEL
LIN {X 0,Y 601.423,Z 81.189,A -85,B 0,C 180,E1 -683.735,E2 -683.735} C_VEL
LIN {X 0,Y 601.424,Z 81.193,A -85,B 0,C 180,E1 -686.063,E2 -686.063} C_VEL
LIN {X 0,Y 601.422,Z 81.195,A -85,B 0,C 180,E1 -688.543,E2 -688.543} C_VEL
LIN {X 0,Y 601.428,Z 81.188,A -85,B 0,C 180,E1 -691.377,E2 -691.377} C_VEL
LIN {X 0,Y 601.41,Z 81.2,A -85,B 0,C 180,E1 -694.13,E2 -694.13} C_VEL
LIN {X 0,Y 601.415,Z 81.192,A -85,B 0,C 180,E1 -696.593,E2 -696.593} C_VEL
LIN {X 0,Y 601.425,Z 81.191,A -85,B 0,C 180,E1 -699.481,E2 -699.481} C_VEL
LIN {X 0,Y 601.393,Z 81.196,A -85,B 0,C 180,E1 -702.315,E2 -702.315} C_VEL
LIN {X 0,Y 601.413,Z 81.192,A -85,B 0,C 180,E1 -704.412,E2 -704.412} C_VEL
LIN {X 0,Y 601.42,Z 81.191,A -85,B 0,C 180,E1 -707.175,E2 -707.175} C_VEL
LIN {X 0,Y 601.424,Z 81.194,A -85,B 0,C 180,E1 -709.907,E2 -709.907} C_VEL
LIN {X 0,Y 601.444,Z 81.186,A -85,B 0,C 180,E1 -712.617,E2 -712.617} C_VEL
LIN {X 0,Y 601.43,Z 81.195,A -85,B 0,C 180,E1 -715.31,E2 -715.31} C_VEL
LIN {X 0,Y 601.414,Z 81.191,A -85,B 0,C 180,E1 -717.993,E2 -717.993} C_VEL
LIN {X 0,Y 601.451,Z 81.186,A -85,B 0,C 180,E1 -720.672,E2 -720.672} C_VEL
LIN {X 0,Y 601.43,Z 81.196,A -85,B 0,C 180,E1 -723.352,E2 -723.352} C_VEL
LIN {X 0,Y 601.401,Z 81.191,A -85,B 0,C 180,E1 -726.039,E2 -726.039} C_VEL
LIN {X 0,Y 601.435,Z 81.192,A -85,B 0,C 180,E1 -728.74,E2 -728.74} C_VEL
LIN {X 0,Y 601.429,Z 81.191,A -85,B 0,C 180,E1 -731.46,E2 -731.46} C_VEL
LIN {X 0,Y 601.413,Z 81.19,A -85,B 0,C 180,E1 -734.207,E2 -734.207} C_VEL
LIN {X 0,Y 601.426,Z 81.195,A -85,B 0,C 180,E1 -736.988,E2 -736.988} C_VEL
LIN {X 0,Y 601.4,Z 81.191,A -85,B 0,C 180,E1 -739.811,E2 -739.811} C_VEL
LIN {X 0,Y 601.41,Z 81.2,A -85,B 0,C 180,E1 -742.607,E2 -742.607} C_VEL
LIN {X 0,Y 601.395,Z 81.197,A -85,B 0,C 180,E1 -744.88,E2 -744.88} C_VEL
LIN {X 0,Y 601.42,Z 81.19,A -85,B 0,C 180,E1 -747.869,E2 -747.869} C_VEL
LIN {X 0,Y 601.425,Z 81.194,A -85,B 0,C 180,E1 -750.166,E2 -750.166} C_VEL
LIN {X 0,Y 601.42,Z 81.193,A -85,B 0,C 180,E1 -752.717,E2 -752.717} C_VEL
LIN {X 0,Y 601.388,Z 81.193,A -85,B 0,C 180,E1 -755.113,E2 -755.113} C_VEL
LIN {X 0,Y 601.432,Z 81.188,A -85,B 0,C 180,E1 -757.421,E2 -757.421} C_VEL
LIN {X 0,Y 601.399,Z 81.2,A -85,B 0,C 180,E1 -759.997,E2 -759.997} C_VEL
LIN {X 0,Y 601.405,Z 81.192,A -85,B 0,C 180,E1 -762.672,E2 -762.672} C_VEL
LIN {X 0,Y 601.424,Z 81.191,A -85,B 0,C 180,E1 -765.483,E2 -765.483} C_VEL
LIN {X 0,Y 601.418,Z 81.191,A -85,B 0,C 180,E1 -768.409,E2 -768.409} C_VEL
LIN {X 0,Y 601.435,Z 81.193,A -85,B 0,C 180,E1 -771.53,E2 -771.53} C_VEL
LIN {X 0,Y 601.381,Z 81.195,A -85,B 0,C 180,E1 -774.246,E2 -774.246} C_VEL
LIN {X 0,Y 601.414,Z 81.19,A -85,B 0,C 180,E1 -776.687,E2 -776.687} C_VEL
LIN {X 0,Y 601.412,Z 81.193,A -85,B 0,C 180,E1 -779.059,E2 -779.059} C_VEL
LIN {X 0,Y 601.431,Z 81.197,A -85,B 0,C 180,E1 -781.374,E2 -781.374} C_VEL
LIN {X 0,Y 601.396,Z 81.198,A -85,B 0,C 180,E1 -783.637,E2 -783.637} C_VEL
LIN {X 0,Y 601.427,Z 81.319,A -85,B 0,C 180,E1 -786.18,E2 -786.18} C_VEL
LIN {X 0,Y 601.739,Z 84.499,A -85,B 0,C 180,E1 -786.604,E2 -786.604} C_VEL
LIN {X 0,Y 601.662,Z 107.108,A -85,B 0,C 180,E1 -789.488,E2 -789.488} C_VEL
LIN {X 0,Y 601.583,Z 129.717,A -85,B 0,C 180,E1 -792.318,E2 -792.318} C_VEL
LIN {X 0,Y 601.559,Z 143.681,A -85,B 0,C 180,E1 -794.039,E2 -794.039} C_VEL
LIN {X 0,Y 601.841,Z 149.493,A -85,B 0,C 180,E1 -794.117,E2 -794.117} C_VEL
LIN {X 0,Y 601.711,Z 280.974,A -85,B 0,C 180,E1 -795.721,E2 -795.721} C_VEL
LIN {X 0,Y 601.701,Z 295.545,A -85,B 0,C 180,E1 -796.036,E2 -796.036} C_VEL
LIN {X 0,Y 601.636,Z 309.741,A -85,B 0,C 180,E1 -796.49,E2 -796.49} C_VEL
LIN {X 0,Y 601.6,Z 323.656,A -85,B 0,C 180,E1 -797.091,E2 -797.091} C_VEL
LIN {X 0,Y 601.542,Z 336.112,A -85,B 0,C 180,E1 -797.776,E2 -797.776} C_VEL
LIN {X 0,Y 601.504,Z 347.487,A -85,B 0,C 180,E1 -798.544,E2 -798.544} C_VEL
LIN {X 0,Y 601.482,Z 357.944,A -85,B 0,C 180,E1 -799.396,E2 -799.396} C_VEL
LIN {X 0,Y 601.43,Z 368.344,A -85,B 0,C 180,E1 -800.416,E2 -800.416} C_VEL
LIN {X 0,Y 601.406,Z 376.921,A -85,B 0,C 180,E1 -801.432,E2 -801.432} C_VEL
LIN {X 0,Y 601.392,Z 385.12,A -85,B 0,C 180,E1 -802.615,E2 -802.615} C_VEL
LIN {X 0,Y 601.361,Z 390.757,A -85,B 0,C 180,E1 -803.605,E2 -803.605} C_VEL
LIN {X 0,Y 601.354,Z 395.572,A -85,B 0,C 180,E1 -804.636,E2 -804.636} C_VEL
LIN {X 0,Y 601.345,Z 400.445,A -85,B 0,C 180,E1 -805.98,E2 -805.98} C_VEL
LIN {X 0,Y 601.322,Z 403.833,A -85,B 0,C 180,E1 -807.321,E2 -807.321} C_VEL
LIN {X 0,Y 601.342,Z 405.832,A -85,B 0,C 180,E1 -808.662,E2 -808.662} C_VEL
LIN {X 0,Y 601.333,Z 406.5,A -85,B 0,C 180,E1 -810.001,E2 -810.001} C_VEL
LIN {X 0,Y 601.342,Z 405.83,A -85,B 0,C 180,E1 -811.34,E2 -811.34} C_VEL
LIN {X 0,Y 601.322,Z 403.83,A -85,B 0,C 180,E1 -812.681,E2 -812.681} C_VEL
LIN {X 0,Y 601.345,Z 400.439,A -85,B 0,C 180,E1 -814.022,E2 -814.022} C_VEL
LIN {X 0,Y 601.355,Z 395.564,A -85,B 0,C 180,E1 -815.366,E2 -815.366} C_VEL
LIN {X 0,Y 601.374,Z 389.621,A -85,B 0,C 180,E1 -816.605,E2 -816.605} C_VEL
LIN {X 0,Y 601.387,Z 382.913,A -85,B 0,C 180,E1 -817.724,E2 -817.724} C_VEL
LIN {X 0,Y 601.412,Z 374.191,A -85,B 0,C 180,E1 -818.908,E2 -818.908} C_VEL
LIN {X 0,Y 601.433,Z 365.073,A -85,B 0,C 180,E1 -819.926,E2 -819.926} C_VEL
LIN {X 0,Y 601.497,Z 354.835,A -85,B 0,C 180,E1 -820.876,E2 -820.876} C_VEL
LIN {X 0,Y 601.535,Z 343.957,A -85,B 0,C 180,E1 -821.713,E2 -821.713} C_VEL
LIN {X 0,Y 601.576,Z 331.761,A -85,B 0,C 180,E1 -822.483,E2 -822.483} C_VEL
LIN {X 0,Y 601.619,Z 320.073,A -85,B 0,C 180,E1 -823.082,E2 -823.082} C_VEL
LIN {X 0,Y 601.657,Z 307.919,A -85,B 0,C 180,E1 -823.579,E2 -823.579} C_VEL
LIN {X 0,Y 601.712,Z 294.026,A -85,B 0,C 180,E1 -824.004,E2 -824.004} C_VEL
LIN {X 0,Y 601.739,Z 279.834,A -85,B 0,C 180,E1 -824.296,E2 -824.296} C_VEL
LIN {X 0,Y 601.742,Z 144.861,A -85,B 0,C 180,E1 -825.942,E2 -825.942} C_VEL
LIN {X 0,Y 601.542,Z 143.478,A -85,B 0,C 180,E1 -825.98,E2 -825.98} C_VEL
LIN {X 0,Y 601.6,Z 122.141,A -85,B 0,C 180,E1 -828.625,E2 -828.625} C_VEL
LIN {X 0,Y 601.701,Z 98.613,A -85,B 0,C 180,E1 -831.589,E2 -831.589} C_VEL
LIN {X 0,Y 601.758,Z 83.07,A -85,B 0,C 180,E1 -833.58,E2 -833.58} C_VEL
LIN {X 0,Y 601.404,Z 81.195,A -85,B 0,C 180,E1 -833.869,E2 -833.869} C_VEL
LIN {X 0,Y 601.399,Z 81.199,A -85,B 0,C 180,E1 -836.365,E2 -836.365} C_VEL
LIN {X 0,Y 601.441,Z 81.192,A -85,B 0,C 180,E1 -838.789,E2 -838.789} C_VEL
LIN {X 0,Y 601.404,Z 81.193,A -85,B 0,C 180,E1 -841.728,E2 -841.728} C_VEL
LIN {X 0,Y 601.425,Z 81.196,A -85,B 0,C 180,E1 -844.119,E2 -844.119} C_VEL
LIN {X 0,Y 601.442,Z 81.187,A -85,B 0,C 180,E1 -847.382,E2 -847.382} C_VEL
LIN {X 0,Y 601.409,Z 81.199,A -85,B 0,C 180,E1 -849.996,E2 -849.996} C_VEL
LIN {X 0,Y 601.414,Z 81.191,A -85,B 0,C 180,E1 -852.671,E2 -852.671} C_VEL
LIN {X 0,Y 601.409,Z 81.194,A -85,B 0,C 180,E1 -855.479,E2 -855.479} C_VEL
LIN {X 0,Y 601.429,Z 81.188,A -85,B 0,C 180,E1 -858.407,E2 -858.407} C_VEL
LIN {X 0,Y 601.406,Z 81.191,A -85,B 0,C 180,E1 -860.872,E2 -860.872} C_VEL
LIN {X 0,Y 601.403,Z 81.199,A -85,B 0,C 180,E1 -863.416,E2 -863.416} C_VEL
LIN {X 0,Y 601.427,Z 81.19,A -85,B 0,C 180,E1 -866.066,E2 -866.066} C_VEL
LIN {X 0,Y 601.428,Z 81.188,A -85,B 0,C 180,E1 -868.545,E2 -868.545} C_VEL
LIN {X 0,Y 601.431,Z 81.196,A -85,B 0,C 180,E1 -871.372,E2 -871.372} C_VEL
LIN {X 0,Y 601.404,Z 81.194,A -85,B 0,C 180,E1 -873.635,E2 -873.635} C_VEL
LIN {X 0,Y 601.454,Z 81.185,A -85,B 0,C 180,E1 -875.858,E2 -875.858} C_VEL
LIN {X 0,Y 601.408,Z 81.197,A -85,B 0,C 180,E1 -878.759,E2 -878.759} C_VEL
LIN {X 0,Y 601.404,Z 81.192,A -85,B 0,C 180,E1 -881.606,E2 -881.606} C_VEL
LIN {X 0,Y 601.417,Z 81.194,A -85,B 0,C 180,E1 -884.407,E2 -884.407} C_VEL
LIN {X 0,Y 601.414,Z 81.192,A -85,B 0,C 180,E1 -887.17,E2 -887.17} C_VEL
LIN {X 0,Y 601.432,Z 81.189,A -85,B 0,C 180,E1 -889.903,E2 -889.903} C_VEL
LIN {X 0,Y 601.41,Z 81.197,A -85,B 0,C 180,E1 -892.613,E2 -892.613} C_VEL
LIN {X 0,Y 601.416,Z 81.189,A -85,B 0,C 180,E1 -895.306,E2 -895.306} C_VEL
LIN {X 0,Y 601.431,Z 81.193,A -85,B 0,C 180,E1 -897.989,E2 -897.989} C_VEL
LIN {X 0,Y 601.434,Z 81.189,A -85,B 0,C 180,E1 -900.667,E2 -900.667} C_VEL
LIN {X 0,Y 601.427,Z 81.189,A -85,B 0,C 180,E1 -903.347,E2 -903.347} C_VEL
LIN {X 0,Y 601.415,Z 81.198,A -85,B 0,C 180,E1 -906.035,E2 -906.035} C_VEL
LIN {X 0,Y 601.435,Z 81.193,A -85,B 0,C 180,E1 -908.058,E2 -908.058} C_VEL
LIN {X 0,Y 601.414,Z 81.19,A -85,B 0,C 180,E1 -911.003,E2 -911.003} C_VEL
LIN {X 0,Y 601.397,Z 81.193,A -85,B 0,C 180,E1 -912.344,E2 -912.344} C_VEL
LIN {X 0,Y 600.726,Z 81.276,A -85,B 0,C 180,E1 -912.904,E2 -912.904} C_VEL
LIN {X 0,Y 597.872,Z 81.638,A -85,B 0,C 180,E1 -913.811,E2 -913.811} C_VEL
LIN {X 0,Y 595.463,Z 81.936,A -85,B 0,C 180,E1 -914.542,E2 -914.542} C_VEL
LIN {X 0,Y 594.429,Z 82.063,A -85,B 0,C 180,E1 -915.105,E2 -915.105} C_VEL
LIN {X 0,Y 594.345,Z 82.073,A -85,B 0,C 180,E1 -915.296,E2 -915.296} C_VEL
LIN {X 0,Y 594.336,Z 82.075,A -85,B 0,C 180,E1 -917.903,E2 -917.903} C_VEL
LIN {X 0,Y 594.391,Z 82.066,A -85,B 0,C 180,E1 -920.773,E2 -920.773} C_VEL
LIN {X 0,Y 594.356,Z 82.072,A -85,B 0,C 180,E1 -923.702,E2 -923.702} C_VEL
LIN {X 0,Y 594.376,Z 82.07,A -85,B 0,C 180,E1 -926.696,E2 -926.696} C_VEL
LIN {X 0,Y 594.369,Z 82.077,A -85,B 0,C 180,E1 -928.995,E2 -928.995} C_VEL
LIN {X 0,Y 594.359,Z 82.07,A -85,B 0,C 180,E1 -931.638,E2 -931.638} C_VEL
LIN {X 0,Y 594.37,Z 82.073,A -85,B 0,C 180,E1 -934.576,E2 -934.576} C_VEL
LIN {X 0,Y 594.368,Z 82.067,A -85,B 0,C 180,E1 -937.605,E2 -937.605} C_VEL
LIN {X 0,Y 594.349,Z 82.08,A -85,B 0,C 180,E1 -940.564,E2 -940.564} C_VEL
LIN {X 0,Y 594.338,Z 82.072,A -85,B 0,C 180,E1 -943.297,E2 -943.297} C_VEL
LIN {X 0,Y 594.338,Z 82.078,A -85,B 0,C 180,E1 -946.158,E2 -946.158} C_VEL
LIN {X 0,Y 594.351,Z 82.077,A -85,B 0,C 180,E1 -948.533,E2 -948.533} C_VEL
LIN {X 0,Y 594.344,Z 82.072,A -85,B 0,C 180,E1 -951.295,E2 -951.295} C_VEL
LIN {X 0,Y 594.37,Z 82.262,A -85,B 0,C 180,E1 -953.068,E2 -953.068} C_VEL
LIN {X 0,Y 594.606,Z 88.281,A -85,B 0,C 180,E1 -953.982,E2 -953.982} C_VEL
LIN {X 0,Y 594.495,Z 104.881,A -85,B 0,C 180,E1 -956.449,E2 -956.449} C_VEL
LIN {X 0,Y 594.479,Z 114.672,A -85,B 0,C 180,E1 -957.89,E2 -957.89} C_VEL
LIN {X 0,Y 595.005,Z 117.805,A -85,B 0,C 180,E1 -957.954,E2 -957.954} C_VEL
LIN {X 0,Y 594.863,Z 251.268,A -85,B 0,C 180,E1 -959.603,E2 -959.603} C_VEL
LIN {X 0,Y 594.8,Z 265.772,A -85,B 0,C 180,E1 -959.923,E2 -959.923} C_VEL
LIN {X 0,Y 594.722,Z 280.075,A -85,B 0,C 180,E1 -960.388,E2 -960.388} C_VEL
LIN {X 0,Y 594.654,Z 293.748,A -85,B 0,C 180,E1 -960.987,E2 -960.987} C_VEL
LIN {X 0,Y 594.581,Z 306.301,A -85,B 0,C 180,E1 -961.687,E2 -961.687} C_VEL
LIN {X 0,Y 594.527,Z 317.298,A -85,B 0,C 180,E1 -962.439,E2 -962.439} C_VEL
LIN {X 0,Y 594.437,Z 328.847,A -85,B 0,C 180,E1 -963.394,E2 -963.394} C_VEL
LIN {X 0,Y 594.37,Z 339.109,A -85,B 0,C 180,E1 -964.431,E2 -964.431} C_VEL
LIN {X 0,Y 594.328,Z 348.349,A -85,B 0,C 180,E1 -965.569,E2 -965.569} C_VEL
LIN {X 0,Y 594.297,Z 355.648,A -85,B 0,C 180,E1 -966.661,E2 -966.661} C_VEL
LIN {X 0,Y 594.286,Z 361.709,A -85,B 0,C 180,E1 -967.763,E2 -967.763} C_VEL
LIN {X 0,Y 594.264,Z 367.49,A -85,B 0,C 180,E1 -969.101,E2 -969.101} C_VEL
LIN {X 0,Y 594.25,Z 371.393,A -85,B 0,C 180,E1 -970.301,E2 -970.301} C_VEL
LIN {X 0,Y 594.243,Z 373.924,A -85,B 0,C 180,E1 -971.377,E2 -971.377} C_VEL
LIN {X 0,Y 594.233,Z 375.941,A -85,B 0,C 180,E1 -972.801,E2 -972.801} C_VEL
LIN {X 0,Y 594.245,Z 376.467,A -85,B 0,C 180,E1 -974.215,E2 -974.215} C_VEL
LIN {X 0,Y 594.24,Z 375.581,A -85,B 0,C 180,E1 -975.618,E2 -975.618} C_VEL
LIN {X 0,Y 594.24,Z 373.289,A -85,B 0,C 180,E1 -977.013,E2 -977.013} C_VEL
LIN {X 0,Y 594.264,Z 369.548,A -85,B 0,C 180,E1 -978.401,E2 -978.401} C_VEL
LIN {X 0,Y 594.259,Z 364.284,A -85,B 0,C 180,E1 -979.781,E2 -979.781} C_VEL
LIN {X 0,Y 594.277,Z 359.182,A -85,B 0,C 180,E1 -980.812,E2 -980.812} C_VEL
LIN {X 0,Y 594.314,Z 351.929,A -85,B 0,C 180,E1 -982.012,E2 -982.012} C_VEL
LIN {X 0,Y 594.382,Z 343.004,A -85,B 0,C 180,E1 -983.209,E2 -983.209} C_VEL
LIN {X 0,Y 594.429,Z 333.689,A -85,B 0,C 180,E1 -984.231,E2 -984.231} C_VEL
LIN {X 0,Y 594.491,Z 322.391,A -85,B 0,C 180,E1 -985.252,E2 -985.252} C_VEL
LIN {X 0,Y 594.553,Z 310.962,A -85,B 0,C 180,E1 -986.102,E2 -986.102} C_VEL
LIN {X 0,Y 594.62,Z 298.342,A -85,B 0,C 180,E1 -986.865,E2 -986.865} C_VEL
LIN {X 0,Y 594.718,Z 286.063,A -85,B 0,C 180,E1 -987.459,E2 -987.459} C_VEL
LIN {X 0,Y 594.78,Z 272.509,A -85,B 0,C 180,E1 -987.968,E2 -987.968} C_VEL
LIN {X 0,Y 594.79,Z 258.459,A -85,B 0,C 180,E1 -988.349,E2 -988.349} C_VEL
LIN {X 0,Y 594.822,Z 243.26,A -85,B 0,C 180,E1 -988.603,E2 -988.603} C_VEL
LIN {X 0,Y 594.876,Z 117.202,A -85,B 0,C 180,E1 -990.147,E2 -990.147} C_VEL
LIN {X 0,Y 594.429,Z 114.612,A -85,B 0,C 180,E1 -990.211,E2 -990.211} C_VEL
LIN {X 0,Y 594.578,Z 96.519,A -85,B 0,C 180,E1 -992.879,E2 -992.879} C_VEL
LIN {X 0,Y 594.53,Z 82.927,A -85,B 0,C 180,E1 -994.915,E2 -994.915} C_VEL
LIN {X 0,Y 594.406,Z 82.067,A -85,B 0,C 180,E1 -995.086,E2 -995.086} C_VEL
LIN {X 0,Y 594.391,Z 82.069,A -85,B 0,C 180,E1 -997.472,E2 -997.472} C_VEL
LIN {X 0,Y 594.392,Z 82.069,A -85,B 0,C 180,E1 -1000.215,E2 -1000.215} C_VEL
LIN {X 0,Y 594.381,Z 82.067,A -85,B 0,C 180,E1 -1002.982,E2 -1002.982} C_VEL
LIN {X 0,Y 594.368,Z 82.075,A -85,B 0,C 180,E1 -1005.78,E2 -1005.78} C_VEL
LIN {X 0,Y 594.379,Z 82.066,A -85,B 0,C 180,E1 -1008.616,E2 -1008.616} C_VEL
LIN {X 0,Y 594.369,Z 82.077,A -85,B 0,C 180,E1 -1011.502,E2 -1011.502} C_VEL
LIN {X 0,Y 594.378,Z 82.071,A -85,B 0,C 180,E1 -1013.703,E2 -1013.703} C_VEL
LIN {X 0,Y 594.373,Z 82.068,A -85,B 0,C 180,E1 -1016.699,E2 -1016.699} C_VEL
LIN {X 0,Y 594.387,Z 82.071,A -85,B 0,C 180,E1 -1018.997,E2 -1018.997} C_VEL
LIN {X 0,Y 594.369,Z 82.07,A -85,B 0,C 180,E1 -1021.649,E2 -1021.649} C_VEL
LIN {X 0,Y 594.369,Z 82.067,A -85,B 0,C 180,E1 -1024.144,E2 -1024.144} C_VEL
LIN {X 0,Y 594.368,Z 82.076,A -85,B 0,C 180,E1 -1027.086,E2 -1027.086} C_VEL
LIN {X 0,Y 594.373,Z 82.067,A -85,B 0,C 180,E1 -1029.78,E2 -1029.78} C_VEL
LIN {X 0,Y 594.364,Z 82.071,A -85,B 0,C 180,E1 -1032.374,E2 -1032.374} C_VEL
LIN {X 0,Y 594.363,Z 82.071,A -85,B 0,C 180,E1 -1035.19,E2 -1035.19} C_VEL
LIN {X 0,Y 594.371,Z 82.069,A -85,B 0,C 180,E1 -1038.151,E2 -1038.151} C_VEL
LIN {X 0,Y 594.377,Z 82.072,A -85,B 0,C 180,E1 -1040.324,E2 -1040.324} C_VEL
LIN {X 0,Y 594.366,Z 82.071,A -85,B 0,C 180,E1 -1042.916,E2 -1042.916} C_VEL
LIN {X 0,Y 594.374,Z 82.069,A -85,B 0,C 180,E1 -1045.86,E2 -1045.86} C_VEL
LIN {X 0,Y 594.372,Z 82.072,A -85,B 0,C 180,E1 -1048.654,E2 -1048.654} C_VEL
LIN {X 0,Y 594.376,Z 82.067,A -85,B 0,C 180,E1 -1051.041,E2 -1051.041} C_VEL
LIN {X 0,Y 594.374,Z 82.067,A -85,B 0,C 180,E1 -1053.303,E2 -1053.303} C_VEL
LIN {X 0,Y 594.384,Z 82.072,A -85,B 0,C 180,E1 -1056.299,E2 -1056.299} C_VEL
LIN {X 0,Y 594.394,Z 82.064,A -85,B 0,C 180,E1 -1059.227,E2 -1059.227} C_VEL
LIN {X 0,Y 594.373,Z 82.074,A -85,B 0,C 180,E1 -1062.099,E2 -1062.099} C_VEL
LIN {X 0,Y 594.365,Z 82.072,A -85,B 0,C 180,E1 -1064.222,E2 -1064.222} C_VEL
LIN {X 0,Y 594.366,Z 82.068,A -85,B 0,C 180,E1 -1067.02,E2 -1067.02} C_VEL
LIN {X 0,Y 594.385,Z 82.073,A -85,B 0,C 180,E1 -1069.787,E2 -1069.787} C_VEL
LIN {X 0,Y 594.408,Z 82.062,A -85,B 0,C 180,E1 -1072.53,E2 -1072.53} C_VEL
LIN {X 0,Y 594.398,Z 82.07,A -85,B 0,C 180,E1 -1075.255,E2 -1075.255} C_VEL
LIN {X 0,Y 594.384,Z 82.067,A -85,B 0,C 180,E1 -1077.969,E2 -1077.969} C_VEL
LIN {X 0,Y 594.421,Z 82.062,A -85,B 0,C 180,E1 -1080.68,E2 -1080.68} C_VEL
LIN {X 0,Y 594.38,Z 82.073,A -85,B 0,C 180,E1 -1083.391,E2 -1083.391} C_VEL
LIN {X 0,Y 594.358,Z 82.068,A -85,B 0,C 180,E1 -1086.111,E2 -1086.111} C_VEL
LIN {X 0,Y 594.395,Z 82.07,A -85,B 0,C 180,E1 -1088.844,E2 -1088.844} C_VEL
LIN {X 0,Y 594.388,Z 82.066,A -85,B 0,C 180,E1 -1091.598,E2 -1091.598} C_VEL
LIN {X 0,Y 594.383,Z 82.068,A -85,B 0,C 180,E1 -1094.379,E2 -1094.379} C_VEL
LIN {X 0,Y 594.384,Z 82.069,A -85,B 0,C 180,E1 -1097.195,E2 -1097.195} C_VEL
LIN {X 0,Y 594.372,Z 82.068,A -85,B 0,C 180,E1 -1100.055,E2 -1100.055} C_VEL
LIN {X 0,Y 594.36,Z 82.073,A -85,B 0,C 180,E1 -1102.969,E2 -1102.969} C_VEL
LIN {X 0,Y 594.371,Z 82.068,A -85,B 0,C 180,E1 -1105.195,E2 -1105.195} C_VEL
LIN {X 0,Y 594.381,Z 82.066,A -85,B 0,C 180,E1 -1107.528,E2 -1107.528} C_VEL
LIN {X 0,Y 594.382,Z 82.075,A -85,B 0,C 180,E1 -1110.33,E2 -1110.33} C_VEL
LIN {X 0,Y 594.376,Z 82.068,A -85,B 0,C 180,E1 -1112.952,E2 -1112.952} C_VEL
LIN {X 0,Y 594.352,Z 82.07,A -85,B 0,C 180,E1 -1115.41,E2 -1115.41} C_VEL
LIN {X 0,Y 594.386,Z 82.071,A -85,B 0,C 180,E1 -1117.942,E2 -1117.942} C_VEL
LIN {X 0,Y 594.374,Z 82.067,A -85,B 0,C 180,E1 -1120.824,E2 -1120.824} C_VEL
LIN {X 0,Y 594.381,Z 82.073,A -85,B 0,C 180,E1 -1123.843,E2 -1123.843} C_VEL
LIN {X 0,Y 594.363,Z 82.068,A -85,B 0,C 180,E1 -1126.702,E2 -1126.702} C_VEL
LIN {X 0,Y 594.37,Z 82.071,A -85,B 0,C 180,E1 -1129.435,E2 -1129.435} C_VEL
LIN {X 0,Y 594.387,Z 82.066,A -85,B 0,C 180,E1 -1132.393,E2 -1132.393} C_VEL
LIN {X 0,Y 594.378,Z 82.073,A -85,B 0,C 180,E1 -1135.421,E2 -1135.421} C_VEL
LIN {X 0,Y 594.375,Z 82.067,A -85,B 0,C 180,E1 -1138.359,E2 -1138.359} C_VEL
LIN {X 0,Y 594.382,Z 82.07,A -85,B 0,C 180,E1 -1141.043,E2 -1141.043} C_VEL
LIN {X 0,Y 594.383,Z 82.075,A -85,B 0,C 180,E1 -1143.302,E2 -1143.302} C_VEL
LIN {X 0,Y 594.411,Z 82.191,A -85,B 0,C 180,E1 -1145.997,E2 -1145.997} C_VEL
LIN {X 0,Y 594.865,Z 85.912,A -85,B 0,C 180,E1 -1146.502,E2 -1146.502} C_VEL
LIN {X 0,Y 594.757,Z 108.521,A -85,B 0,C 180,E1 -1149.419,E2 -1149.419} C_VEL
LIN {X 0,Y 594.599,Z 132.543,A -85,B 0,C 180,E1 -1152.459,E2 -1152.459} C_VEL
LIN {X 0,Y 594.547,Z 143.582,A -85,B 0,C 180,E1 -1153.84,E2 -1153.84} C_VEL
LIN {X 0,Y 595.048,Z 147.705,A -85,B 0,C 180,E1 -1153.909,E2 -1153.909} C_VEL
LIN {X 0,Y 594.855,Z 281.942,A -85,B 0,C 180,E1 -1155.57,E2 -1155.57} C_VEL
LIN {X 0,Y 594.808,Z 296.223,A -85,B 0,C 180,E1 -1155.891,E2 -1155.891} C_VEL
LIN {X 0,Y 594.715,Z 309.741,A -85,B 0,C 180,E1 -1156.33,E2 -1156.33} C_VEL
LIN {X 0,Y 594.646,Z 323.66,A -85,B 0,C 180,E1 -1156.937,E2 -1156.937} C_VEL
LIN {X 0,Y 594.58,Z 336.114,A -85,B 0,C 180,E1 -1157.63,E2 -1157.63} C_VEL
LIN {X 0,Y 594.523,Z 348.574,A -85,B 0,C 180,E1 -1158.489,E2 -1158.489} C_VEL
LIN {X 0,Y 594.448,Z 359.847,A -85,B 0,C 180,E1 -1159.442,E2 -1159.442} C_VEL
LIN {X 0,Y 594.368,Z 369.859,A -85,B 0,C 180,E1 -1160.472,E2 -1160.472} C_VEL
LIN {X 0,Y 594.323,Z 378.178,A -85,B 0,C 180,E1 -1161.501,E2 -1161.501} C_VEL
LIN {X 0,Y 594.303,Z 386.132,A -85,B 0,C 180,E1 -1162.698,E2 -1162.698} C_VEL
LIN {X 0,Y 594.281,Z 392.532,A -85,B 0,C 180,E1 -1163.891,E2 -1163.891} C_VEL
LIN {X 0,Y 594.236,Z 398.203,A -85,B 0,C 180,E1 -1165.252,E2 -1165.252} C_VEL
LIN {X 0,Y 594.258,Z 402.318,A -85,B 0,C 180,E1 -1166.611,E2 -1166.611} C_VEL
LIN {X 0,Y 594.242,Z 405.002,A -85,B 0,C 180,E1 -1167.968,E2 -1167.968} C_VEL
LIN {X 0,Y 594.234,Z 406.333,A -85,B 0,C 180,E1 -1169.323,E2 -1169.323} C_VEL
LIN {X 0,Y 594.234,Z 406.332,A -85,B 0,C 180,E1 -1170.679,E2 -1170.679} C_VEL
LIN {X 0,Y 594.242,Z 404.999,A -85,B 0,C 180,E1 -1172.034,E2 -1172.034} C_VEL
LIN {X 0,Y 594.258,Z 402.314,A -85,B 0,C 180,E1 -1173.391,E2 -1173.391} C_VEL
LIN {X 0,Y 594.236,Z 398.196,A -85,B 0,C 180,E1 -1174.75,E2 -1174.75} C_VEL
LIN {X 0,Y 594.281,Z 392.522,A -85,B 0,C 180,E1 -1176.111,E2 -1176.111} C_VEL
LIN {X 0,Y 594.304,Z 386.12,A -85,B 0,C 180,E1 -1177.304,E2 -1177.304} C_VEL
LIN {X 0,Y 594.324,Z 378.164,A -85,B 0,C 180,E1 -1178.501,E2 -1178.501} C_VEL
LIN {X 0,Y 594.368,Z 369.842,A -85,B 0,C 180,E1 -1179.53,E2 -1179.53} C_VEL
LIN {X 0,Y 594.449,Z 359.826,A -85,B 0,C 180,E1 -1180.56,E2 -1180.56} C_VEL
LIN {X 0,Y 594.494,Z 348.553,A -85,B 0,C 180,E1 -1181.514,E2 -1181.514} C_VEL
LIN {X 0,Y 594.581,Z 336.083,A -85,B 0,C 180,E1 -1182.372,E2 -1182.372} C_VEL
LIN {X 0,Y 594.646,Z 323.621,A -85,B 0,C 180,E1 -1183.065,E2 -1183.065} C_VEL
LIN {X 0,Y 594.714,Z 309.686,A -85,B 0,C 180,E1 -1183.672,E2 -1183.672} C_VEL
LIN {X 0,Y 594.796,Z 295.59,A -85,B 0,C 180,E1 -1184.128,E2 -1184.128} C_VEL
LIN {X 0,Y 594.854,Z 281.836,A -85,B 0,C 180,E1 -1184.432,E2 -1184.432} C_VEL
LIN {X 0,Y 594.925,Z 145.753,A -85,B 0,C 180,E1 -1186.119,E2 -1186.119} C_VEL
LIN {X 0,Y 594.524,Z 143.478,A -85,B 0,C 180,E1 -1186.174,E2 -1186.174} C_VEL
LIN {X 0,Y 594.653,Z 121.908,A -85,B 0,C 180,E1 -1188.88,E2 -1188.88} C_VEL
LIN {X 0,Y 594.79,Z 100.026,A -85,B 0,C 180,E1 -1191.67,E2 -1191.67} C_VEL
LIN {X 0,Y 594.85,Z 84.483,A -85,B 0,C 180,E1 -1193.685,E2 -1193.685} C_VEL
LIN {X 0,Y 594.383,Z 82.072,A -85,B 0,C 180,E1 -1194.029,E2 -1194.029} C_VEL
LIN {X 0,Y 594.386,Z 82.074,A -85,B 0,C 180,E1 -1196.7,E2 -1196.7} C_VEL
LIN {X 0,Y 594.387,Z 82.068,A -85,B 0,C 180,E1 -1198.999,E2 -1198.999} C_VEL
LIN {X 0,Y 594.381,Z 82.067,A -85,B 0,C 180,E1 -1201.642,E2 -1201.642} C_VEL
LIN {X 0,Y 594.382,Z 82.071,A -85,B 0,C 180,E1 -1204.581,E2 -1204.581} C_VEL
LIN {X 0,Y 594.397,Z 82.066,A -85,B 0,C 180,E1 -1207.608,E2 -1207.608} C_VEL
LIN {X 0,Y 594.374,Z 82.069,A -85,B 0,C 180,E1 -1210.568,E2 -1210.568} C_VEL
LIN {X 0,Y 594.36,Z 82.07,A -85,B 0,C 180,E1 -1213.301,E2 -1213.301} C_VEL
LIN {X 0,Y 594.372,Z 82.072,A -85,B 0,C 180,E1 -1216.161,E2 -1216.161} C_VEL
LIN {X 0,Y 594.386,Z 82.064,A -85,B 0,C 180,E1 -1218.535,E2 -1218.535} C_VEL
LIN {X 0,Y 594.379,Z 82.071,A -85,B 0,C 180,E1 -1221.297,E2 -1221.297} C_VEL
LIN {X 0,Y 594.358,Z 82.075,A -85,B 0,C 180,E1 -1223.755,E2 -1223.755} C_VEL
LIN {X 0,Y 594.374,Z 82.067,A -85,B 0,C 180,E1 -1226.237,E2 -1226.237} C_VEL
LIN {X 0,Y 594.375,Z 82.067,A -85,B 0,C 180,E1 -1228.649,E2 -1228.649} C_VEL
LIN {X 0,Y 594.389,Z 82.071,A -85,B 0,C 180,E1 -1231.043,E2 -1231.043} C_VEL
LIN {X 0,Y 594.387,Z 82.073,A -85,B 0,C 180,E1 -1233.299,E2 -1233.299} C_VEL
LIN {X 0,Y 594.379,Z 82.066,A -85,B 0,C 180,E1 -1236.294,E2 -1236.294} C_VEL
LIN {X 0,Y 594.402,Z 82.068,A -85,B 0,C 180,E1 -1239.223,E2 -1239.223} C_VEL
LIN {X 0,Y 594.353,Z 82.07,A -85,B 0,C 180,E1 -1242.093,E2 -1242.093} C_VEL
LIN {X 0,Y 594.369,Z 82.069,A -85,B 0,C 180,E1 -1244.217,E2 -1244.217} C_VEL
LIN {X 0,Y 594.386,Z 82.07,A -85,B 0,C 180,E1 -1246.319,E2 -1246.319} C_VEL
LIN {X 0,Y 594.37,Z 82.069,A -85,B 0,C 180,E1 -1249.093,E2 -1249.093} C_VEL
LIN {X 0,Y 594.387,Z 82.066,A -85,B 0,C 180,E1 -1251.841,E2 -1251.841} C_VEL
LIN {X 0,Y 594.383,Z 82.072,A -85,B 0,C 180,E1 -1254.57,E2 -1254.57} C_VEL
LIN {X 0,Y 594.405,Z 82.062,A -85,B 0,C 180,E1 -1257.287,E2 -1257.287} C_VEL
LIN {X 0,Y 594.421,Z 82.068,A -85,B 0,C 180,E1 -1259.998,E2 -1259.998} C_VEL
LIN {X 0,Y 594.392,Z 82.066,A -85,B 0,C 180,E1 -1262.709,E2 -1262.709} C_VEL
LIN {X 0,Y 594.396,Z 82.066,A -85,B 0,C 180,E1 -1265.425,E2 -1265.425} C_VEL
LIN {X 0,Y 594.38,Z 82.07,A -85,B 0,C 180,E1 -1268.155,E2 -1268.155} C_VEL
LIN {X 0,Y 594.379,Z 82.067,A -85,B 0,C 180,E1 -1271.065,E2 -1271.065} C_VEL
LIN {X 0,Y 594.371,Z 82.076,A -85,B 0,C 180,E1 -1273.676,E2 -1273.676} C_VEL
LIN {X 0,Y 594.345,Z 82.073,A -85,B 0,C 180,E1 -1275.296,E2 -1275.296} C_VEL
LIN {X 0,Y 593.673,Z 82.16,A -85,B 0,C 180,E1 -1275.862,E2 -1275.862} C_VEL
LIN {X 0,Y 590.805,Z 82.515,A -85,B 0,C 180,E1 -1276.78,E2 -1276.78} C_VEL
LIN {X 0,Y 588.392,Z 82.822,A -85,B 0,C 180,E1 -1277.518,E2 -1277.518} C_VEL
LIN {X 0,Y 587.369,Z 82.942,A -85,B 0,C 180,E1 -1278.088,E2 -1278.088} C_VEL
LIN {X 0,Y 587.293,Z 82.949,A -85,B 0,C 180,E1 -1278.281,E2 -1278.281} C_VEL
LIN {X 0,Y 587.327,Z 82.949,A -85,B 0,C 180,E1 -1281.035,E2 -1281.035} C_VEL
LIN {X 0,Y 587.303,Z 82.957,A -85,B 0,C 180,E1 -1283.256,E2 -1283.256} C_VEL
LIN {X 0,Y 587.316,Z 82.95,A -85,B 0,C 180,E1 -1285.514,E2 -1285.514} C_VEL
LIN {X 0,Y 587.33,Z 82.945,A -85,B 0,C 180,E1 -1287.815,E2 -1287.815} C_VEL
LIN {X 0,Y 587.31,Z 82.948,A -85,B 0,C 180,E1 -1290.504,E2 -1290.504} C_VEL
LIN {X 0,Y 587.323,Z 82.95,A -85,B 0,C 180,E1 -1293.108,E2 -1293.108} C_VEL
LIN {X 0,Y 587.275,Z 82.952,A -85,B 0,C 180,E1 -1295.897,E2 -1295.897} C_VEL
LIN {X 0,Y 587.302,Z 82.954,A -85,B 0,C 180,E1 -1298.477,E2 -1298.477} C_VEL
LIN {X 0,Y 587.311,Z 82.949,A -85,B 0,C 180,E1 -1301.154,E2 -1301.154} C_VEL
LIN {X 0,Y 587.297,Z 82.953,A -85,B 0,C 180,E1 -1304.109,E2 -1304.109} C_VEL
LIN {X 0,Y 587.271,Z 82.954,A -85,B 0,C 180,E1 -1306.989,E2 -1306.989} C_VEL
LIN {X 0,Y 587.284,Z 82.955,A -85,B 0,C 180,E1 -1309.742,E2 -1309.742} C_VEL
LIN {X 0,Y 587.315,Z 82.954,A -85,B 0,C 180,E1 -1312.389,E2 -1312.389} C_VEL
LIN {X 0,Y 587.338,Z 83.08,A -85,B 0,C 180,E1 -1312.93,E2 -1312.93} C_VEL
LIN {X 0,Y 587.666,Z 88.062,A -85,B 0,C 180,E1 -1313.702,E2 -1313.702} C_VEL
LIN {X 0,Y 587.548,Z 104.687,A -85,B 0,C 180,E1 -1316.205,E2 -1316.205} C_VEL
LIN {X 0,Y 587.469,Z 114.655,A -85,B 0,C 180,E1 -1317.689,E2 -1317.689} C_VEL
LIN {X 0,Y 588.193,Z 119.386,A -85,B 0,C 180,E1 -1317.782,E2 -1317.782} C_VEL
LIN {X 0,Y 588.01,Z 251.005,A -85,B 0,C 180,E1 -1319.426,E2 -1319.426} C_VEL
LIN {X 0,Y 587.924,Z 265.216,A -85,B 0,C 180,E1 -1319.738,E2 -1319.738} C_VEL
LIN {X 0,Y 587.854,Z 278.267,A -85,B 0,C 180,E1 -1320.155,E2 -1320.155} C_VEL
LIN {X 0,Y 587.754,Z 291.464,A -85,B 0,C 180,E1 -1320.717,E2 -1320.717} C_VEL
LIN {X 0,Y 587.638,Z 304.375,A -85,B 0,C 180,E1 -1321.419,E2 -1321.419} C_VEL
LIN {X 0,Y 587.544,Z 316.823,A -85,B 0,C 180,E1 -1322.263,E2 -1322.263} C_VEL
LIN {X 0,Y 587.451,Z 327.569,A -85,B 0,C 180,E1 -1323.151,E2 -1323.151} C_VEL
LIN {X 0,Y 587.348,Z 337.167,A -85,B 0,C 180,E1 -1324.103,E2 -1324.103} C_VEL
LIN {X 0,Y 587.307,Z 346.675,A -85,B 0,C 180,E1 -1325.239,E2 -1325.239} C_VEL
LIN {X 0,Y 587.245,Z 354.399,A -85,B 0,C 180,E1 -1326.363,E2 -1326.363} C_VEL
LIN {X 0,Y 587.182,Z 360.67,A -85,B 0,C 180,E1 -1327.479,E2 -1327.479} C_VEL
LIN {X 0,Y 587.205,Z 365.726,A -85,B 0,C 180,E1 -1328.589,E2 -1328.589} C_VEL
LIN {X 0,Y 587.178,Z 369.711,A -85,B 0,C 180,E1 -1329.689,E2 -1329.689} C_VEL
LIN {X 0,Y 587.146,Z 373.505,A -85,B 0,C 180,E1 -1331.144,E2 -1331.144} C_VEL
LIN {X 0,Y 587.121,Z 375.734,A -85,B 0,C 180,E1 -1332.586,E2 -1332.586} C_VEL
LIN {X 0,Y 587.15,Z 376.499,A -85,B 0,C 180,E1 -1334.019,E2 -1334.019} C_VEL
LIN {X 0,Y 587.155,Z 375.805,A -85,B 0,C 180,E1 -1335.441,E2 -1335.441} C_VEL
LIN {X 0,Y 587.14,Z 373.698,A -85,B 0,C 180,E1 -1336.853,E2 -1336.853} C_VEL
LIN {X 0,Y 587.17,Z 370.149,A -85,B 0,C 180,E1 -1338.259,E2 -1338.259} C_VEL
LIN {X 0,Y 587.191,Z 366.525,A -85,B 0,C 180,E1 -1339.308,E2 -1339.308} C_VEL
LIN {X 0,Y 587.203,Z 361.945,A -85,B 0,C 180,E1 -1340.353,E2 -1340.353} C_VEL
LIN {X 0,Y 587.223,Z 355.358,A -85,B 0,C 180,E1 -1341.569,E2 -1341.569} C_VEL
LIN {X 0,Y 587.269,Z 347.224,A -85,B 0,C 180,E1 -1342.78,E2 -1342.78} C_VEL
LIN {X 0,Y 587.326,Z 338.754,A -85,B 0,C 180,E1 -1343.817,E2 -1343.817} C_VEL
LIN {X 0,Y 587.43,Z 328.55,A -85,B 0,C 180,E1 -1344.851,E2 -1344.851} C_VEL
LIN {X 0,Y 587.517,Z 317.227,A -85,B 0,C 180,E1 -1345.797,E2 -1345.797} C_VEL
LIN {X 0,Y 587.609,Z 304.623,A -85,B 0,C 180,E1 -1346.656,E2 -1346.656} C_VEL
LIN {X 0,Y 587.718,Z 292.087,A -85,B 0,C 180,E1 -1347.343,E2 -1347.343} C_VEL
LIN {X 0,Y 587.84,Z 278.061,A -85,B 0,C 180,E1 -1347.944,E2 -1347.944} C_VEL
LIN {X 0,Y 587.923,Z 263.663,A -85,B 0,C 180,E1 -1348.394,E2 -1348.394} C_VEL
LIN {X 0,Y 587.966,Z 249.111,A -85,B 0,C 180,E1 -1348.693,E2 -1348.693} C_VEL
LIN {X 0,Y 588.034,Z 117.92,A -85,B 0,C 180,E1 -1350.331,E2 -1350.331} C_VEL
LIN {X 0,Y 587.446,Z 114.627,A -85,B 0,C 180,E1 -1350.406,E2 -1350.406} C_VEL
LIN {X 0,Y 587.626,Z 95.552,A -85,B 0,C 180,E1 -1353.256,E2 -1353.256} C_VEL
LIN {X 0,Y 587.564,Z 84.242,A -85,B 0,C 180,E1 -1354.974,E2 -1354.974} C_VEL
LIN {X 0,Y 587.379,Z 82.944,A -85,B 0,C 180,E1 -1355.191,E2 -1355.191} C_VEL
LIN {X 0,Y 587.354,Z 82.947,A -85,B 0,C 180,E1 -1357.562,E2 -1357.562} C_VEL
LIN {X 0,Y 587.337,Z 82.946,A -85,B 0,C 180,E1 -1360.339,E2 -1360.339} C_VEL
LIN {X 0,Y 587.327,Z 82.947,A -85,B 0,C 180,E1 -1363.14,E2 -1363.14} C_VEL
LIN {X 0,Y 587.337,Z 82.947,A -85,B 0,C 180,E1 -1365.262,E2 -1365.262} C_VEL
LIN {X 0,Y 587.336,Z 82.95,A -85,B 0,C 180,E1 -1367.405,E2 -1367.405} C_VEL
LIN {X 0,Y 587.325,Z 82.954,A -85,B 0,C 180,E1 -1369.574,E2 -1369.574} C_VEL
LIN {X 0,Y 587.343,Z 82.942,A -85,B 0,C 180,E1 -1372.512,E2 -1372.512} C_VEL
LIN {X 0,Y 587.321,Z 82.952,A -85,B 0,C 180,E1 -1375.516,E2 -1375.516} C_VEL
LIN {X 0,Y 587.321,Z 82.947,A -85,B 0,C 180,E1 -1377.818,E2 -1377.818} C_VEL
LIN {X 0,Y 587.332,Z 82.945,A -85,B 0,C 180,E1 -1380.517,E2 -1380.517} C_VEL
LIN {X 0,Y 587.325,Z 82.95,A -85,B 0,C 180,E1 -1383.396,E2 -1383.396} C_VEL
LIN {X 0,Y 587.333,Z 82.944,A -85,B 0,C 180,E1 -1385.896,E2 -1385.896} C_VEL
LIN {X 0,Y 587.318,Z 82.948,A -85,B 0,C 180,E1 -1388.479,E2 -1388.479} C_VEL
LIN {X 0,Y 587.336,Z 82.949,A -85,B 0,C 180,E1 -1391.155,E2 -1391.155} C_VEL
LIN {X 0,Y 587.303,Z 82.949,A -85,B 0,C 180,E1 -1394.116,E2 -1394.116} C_VEL
LIN {X 0,Y 587.317,Z 82.951,A -85,B 0,C 180,E1 -1396.999,E2 -1396.999} C_VEL
LIN {X 0,Y 587.305,Z 82.947,A -85,B 0,C 180,E1 -1399.75,E2 -1399.75} C_VEL
LIN {X 0,Y 587.325,Z 82.953,A -85,B 0,C 180,E1 -1402.395,E2 -1402.395} C_VEL
LIN {X 0,Y 587.333,Z 82.946,A -85,B 0,C 180,E1 -1404.949,E2 -1404.949} C_VEL
LIN {X 0,Y 587.326,Z 82.945,A -85,B 0,C 180,E1 -1407.424,E2 -1407.424} C_VEL
LIN {X 0,Y 587.326,Z 82.948,A -85,B 0,C 180,E1 -1409.833,E2 -1409.833} C_VEL
LIN {X 0,Y 587.328,Z 82.953,A -85,B 0,C 180,E1 -1412.309,E2 -1412.309} C_VEL
LIN {X 0,Y 587.328,Z 82.949,A -85,B 0,C 180,E1 -1414.487,E2 -1414.487} C_VEL
LIN {X 0,Y 587.351,Z 82.943,A -85,B 0,C 180,E1 -1417.49,E2 -1417.49} C_VEL
LIN {X 0,Y 587.331,Z 82.947,A -85,B 0,C 180,E1 -1420.428,E2 -1420.428} C_VEL
LIN {X 0,Y 587.341,Z 82.945,A -85,B 0,C 180,E1 -1423.314,E2 -1423.314} C_VEL
LIN {X 0,Y 587.348,Z 82.946,A -85,B 0,C 180,E1 -1426.157,E2 -1426.157} C_VEL
LIN {X 0,Y 587.335,Z 82.944,A -85,B 0,C 180,E1 -1428.965,E2 -1428.965} C_VEL
LIN {X 0,Y 587.361,Z 82.948,A -85,B 0,C 180,E1 -1431.747,E2 -1431.747} C_VEL
LIN {X 0,Y 587.355,Z 82.941,A -85,B 0,C 180,E1 -1434.509,E2 -1434.509} C_VEL
LIN {X 0,Y 587.377,Z 82.945,A -85,B 0,C 180,E1 -1437.259,E2 -1437.259} C_VEL
LIN {X 0,Y 587.37,Z 82.94,A -85,B 0,C 180,E1 -1440.002,E2 -1440.002} C_VEL
LIN {X 0,Y 587.374,Z 82.941,A -85,B 0,C 180,E1 -1442.745,E2 -1442.745} C_VEL
LIN {X 0,Y 587.354,Z 82.946,A -85,B 0,C 180,E1 -1445.495,E2 -1445.495} C_VEL
LIN {X 0,Y 587.362,Z 82.94,A -85,B 0,C 180,E1 -1448.257,E2 -1448.257} C_VEL
LIN {X 0,Y 587.34,Z 82.951,A -85,B 0,C 180,E1 -1451.136,E2 -1451.136} C_VEL
LIN {X 0,Y 587.358,Z 82.942,A -85,B 0,C 180,E1 -1454.263,E2 -1454.263} C_VEL
LIN {X 0,Y 587.346,Z 82.944,A -85,B 0,C 180,E1 -1457.408,E2 -1457.408} C_VEL
LIN {X 0,Y 587.327,Z 82.948,A -85,B 0,C 180,E1 -1460.307,E2 -1460.307} C_VEL
LIN {X 0,Y 587.319,Z 82.947,A -85,B 0,C 180,E1 -1463.26,E2 -1463.26} C_VEL
LIN {X 0,Y 587.333,Z 82.944,A -85,B 0,C 180,E1 -1465.518,E2 -1465.518} C_VEL
LIN {X 0,Y 587.346,Z 82.943,A -85,B 0,C 180,E1 -1467.819,E2 -1467.819} C_VEL
LIN {X 0,Y 587.331,Z 82.952,A -85,B 0,C 180,E1 -1470.511,E2 -1470.511} C_VEL
LIN {X 0,Y 587.334,Z 82.944,A -85,B 0,C 180,E1 -1473.398,E2 -1473.398} C_VEL
LIN {X 0,Y 587.315,Z 82.951,A -85,B 0,C 180,E1 -1475.9,E2 -1475.9} C_VEL
LIN {X 0,Y 587.327,Z 82.949,A -85,B 0,C 180,E1 -1478.481,E2 -1478.481} C_VEL
LIN {X 0,Y 587.335,Z 82.943,A -85,B 0,C 180,E1 -1481.158,E2 -1481.158} C_VEL
LIN {X 0,Y 587.333,Z 82.951,A -85,B 0,C 180,E1 -1484.116,E2 -1484.116} C_VEL
LIN {X 0,Y 587.312,Z 82.946,A -85,B 0,C 180,E1 -1486.995,E2 -1486.995} C_VEL
LIN {X 0,Y 587.312,Z 82.956,A -85,B 0,C 180,E1 -1489.747,E2 -1489.747} C_VEL
LIN {X 0,Y 587.343,Z 82.944,A -85,B 0,C 180,E1 -1492.394,E2 -1492.394} C_VEL
LIN {X 0,Y 587.342,Z 82.953,A -85,B 0,C 180,E1 -1495.654,E2 -1495.654} C_VEL
LIN {X 0,Y 587.34,Z 82.944,A -85,B 0,C 180,E1 -1498.232,E2 -1498.232} C_VEL
LIN {X 0,Y 587.347,Z 82.945,A -85,B 0,C 180,E1 -1500.868,E2 -1500.868} C_VEL
LIN {X 0,Y 587.335,Z 82.95,A -85,B 0,C 180,E1 -1503.723,E2 -1503.723} C_VEL
LIN {X 0,Y 587.38,Z 83.107,A -85,B 0,C 180,E1 -1505.831,E2 -1505.831} C_VEL
LIN {X 0,Y 587.982,Z 87.232,A -85,B 0,C 180,E1 -1506.397,E2 -1506.397} C_VEL
LIN {X 0,Y 587.855,Z 109.934,A -85,B 0,C 180,E1 -1509.35,E2 -1509.35} C_VEL
LIN {X 0,Y 587.63,Z 133.956,A -85,B 0,C 180,E1 -1512.424,E2 -1512.424} C_VEL
LIN {X 0,Y 587.554,Z 143.582,A -85,B 0,C 180,E1 -1513.642,E2 -1513.642} C_VEL
LIN {X 0,Y 588.224,Z 147.705,A -85,B 0,C 180,E1 -1513.717,E2 -1513.717} C_VEL
LIN {X 0,Y 587.992,Z 281.941,A -85,B 0,C 180,E1 -1515.398,E2 -1515.398} C_VEL
LIN {X 0,Y 587.925,Z 296.337,A -85,B 0,C 180,E1 -1515.725,E2 -1515.725} C_VEL
LIN {X 0,Y 587.801,Z 310.867,A -85,B 0,C 180,E1 -1516.21,E2 -1516.21} C_VEL
LIN {X 0,Y 587.725,Z 323.663,A -85,B 0,C 180,E1 -1516.781,E2 -1516.781} C_VEL
LIN {X 0,Y 587.604,Z 336.116,A -85,B 0,C 180,E1 -1517.481,E2 -1517.481} C_VEL
LIN {X 0,Y 587.512,Z 347.493,A -85,B 0,C 180,E1 -1518.268,E2 -1518.268} C_VEL
LIN {X 0,Y 587.465,Z 357.946,A -85,B 0,C 180,E1 -1519.14,E2 -1519.14} C_VEL
LIN {X 0,Y 587.353,Z 368.343,A -85,B 0,C 180,E1 -1520.184,E2 -1520.184} C_VEL
LIN {X 0,Y 587.311,Z 376.92,A -85,B 0,C 180,E1 -1521.225,E2 -1521.225} C_VEL
LIN {X 0,Y 587.249,Z 385.121,A -85,B 0,C 180,E1 -1522.436,E2 -1522.436} C_VEL
LIN {X 0,Y 587.18,Z 391.687,A -85,B 0,C 180,E1 -1523.637,E2 -1523.637} C_VEL
LIN {X 0,Y 587.158,Z 396.965,A -85,B 0,C 180,E1 -1524.851,E2 -1524.851} C_VEL
LIN {X 0,Y 587.181,Z 400.446,A -85,B 0,C 180,E1 -1525.883,E2 -1525.883} C_VEL
LIN {X 0,Y 587.129,Z 403.834,A -85,B 0,C 180,E1 -1527.257,E2 -1527.257} C_VEL
LIN {X 0,Y 587.142,Z 405.833,A -85,B 0,C 180,E1 -1528.629,E2 -1528.629} C_VEL
LIN {X 0,Y 587.135,Z 406.5,A -85,B 0,C 180,E1 -1530.001,E2 -1530.001} C_VEL
LIN {X 0,Y 587.142,Z 405.832,A -85,B 0,C 180,E1 -1531.373,E2 -1531.373} C_VEL
LIN {X 0,Y 587.129,Z 403.831,A -85,B 0,C 180,E1 -1532.745,E2 -1532.745} C_VEL
LIN {X 0,Y 587.181,Z 400.441,A -85,B 0,C 180,E1 -1534.119,E2 -1534.119} C_VEL
LIN {X 0,Y 587.2,Z 395.564,A -85,B 0,C 180,E1 -1535.495,E2 -1535.495} C_VEL
LIN {X 0,Y 587.211,Z 389.048,A -85,B 0,C 180,E1 -1536.875,E2 -1536.875} C_VEL
LIN {X 0,Y 587.269,Z 381.794,A -85,B 0,C 180,E1 -1538.084,E2 -1538.084} C_VEL
LIN {X 0,Y 587.322,Z 372.815,A -85,B 0,C 180,E1 -1539.297,E2 -1539.297} C_VEL
LIN {X 0,Y 587.372,Z 363.382,A -85,B 0,C 180,E1 -1540.34,E2 -1540.34} C_VEL
LIN {X 0,Y 587.473,Z 353.025,A -85,B 0,C 180,E1 -1541.291,E2 -1541.291} C_VEL
LIN {X 0,Y 587.574,Z 341.419,A -85,B 0,C 180,E1 -1542.171,E2 -1542.171} C_VEL
LIN {X 0,Y 587.665,Z 328.629,A -85,B 0,C 180,E1 -1542.959,E2 -1542.959} C_VEL
LIN {X 0,Y 587.788,Z 316.135,A -85,B 0,C 180,E1 -1543.572,E2 -1543.572} C_VEL
LIN {X 0,Y 587.899,Z 302.701,A -85,B 0,C 180,E1 -1544.082,E2 -1544.082} C_VEL
LIN {X 0,Y 587.966,Z 288.264,A -85,B 0,C 180,E1 -1544.478,E2 -1544.478} C_VEL
LIN {X 0,Y 588.011,Z 274.533,A -85,B 0,C 180,E1 -1544.714,E2 -1544.714} C_VEL
LIN {X 0,Y 588.174,Z 146.983,A -85,B 0,C 180,E1 -1546.293,E2 -1546.293} C_VEL
LIN {X 0,Y 587.574,Z 143.478,A -85,B 0,C 180,E1 -1546.37,E2 -1546.37} C_VEL
LIN {X 0,Y 587.71,Z 122.64,A -85,B 0,C 180,E1 -1549.018,E2 -1549.018} C_VEL
LIN {X 0,Y 587.901,Z 101.439,A -85,B 0,C 180,E1 -1551.753,E2 -1551.753} C_VEL
LIN {X 0,Y 587.903,Z 85.757,A -85,B 0,C 180,E1 -1553.796,E2 -1553.796} C_VEL
LIN {X 0,Y 587.351,Z 82.95,A -85,B 0,C 180,E1 -1554.213,E2 -1554.213} C_VEL
LIN {X 0,Y 587.335,Z 82.947,A -85,B 0,C 180,E1 -1557.047,E2 -1557.047} C_VEL
LIN {X 0,Y 587.347,Z 82.943,A -85,B 0,C 180,E1 -1559.38,E2 -1559.38} C_VEL
LIN {X 0,Y 587.349,Z 82.945,A -85,B 0,C 180,E1 -1561.835,E2 -1561.835} C_VEL
LIN {X 0,Y 587.348,Z 82.951,A -85,B 0,C 180,E1 -1564.347,E2 -1564.347} C_VEL
LIN {X 0,Y 587.352,Z 82.943,A -85,B 0,C 180,E1 -1567.608,E2 -1567.608} C_VEL
LIN {X 0,Y 587.319,Z 82.952,A -85,B 0,C 180,E1 -1570.255,E2 -1570.255} C_VEL
LIN {X 0,Y 587.312,Z 82.947,A -85,B 0,C 180,E1 -1573.117,E2 -1573.117} C_VEL
LIN {X 0,Y 587.324,Z 82.952,A -85,B 0,C 180,E1 -1576.048,E2 -1576.048} C_VEL
LIN {X 0,Y 587.343,Z 82.941,A -85,B 0,C 180,E1 -1578.925,E2 -1578.925} C_VEL
LIN {X 0,Y 587.328,Z 82.953,A -85,B 0,C 180,E1 -1581.519,E2 -1581.519} C_VEL
LIN {X 0,Y 587.299,Z 82.95,A -85,B 0,C 180,E1 -1584.099,E2 -1584.099} C_VEL
LIN {X 0,Y 587.347,Z 82.944,A -85,B 0,C 180,E1 -1586.888,E2 -1586.888} C_VEL
LIN {X 0,Y 587.333,Z 82.951,A -85,B 0,C 180,E1 -1589.492,E2 -1589.492} C_VEL
LIN {X 0,Y 587.317,Z 82.945,A -85,B 0,C 180,E1 -1592.179,E2 -1592.179} C_VEL
LIN {X 0,Y 587.359,Z 82.947,A -85,B 0,C 180,E1 -1595.24,E2 -1595.24} C_VEL
LIN {X 0,Y 587.322,Z 82.946,A -85,B 0,C 180,E1 -1598.224,E2 -1598.224} C_VEL
LIN {X 0,Y 587.35,Z 82.947,A -85,B 0,C 180,E1 -1601.15,E2 -1601.15} C_VEL
LIN {X 0,Y 587.323,Z 82.945,A -85,B 0,C 180,E1 -1604.023,E2 -1604.023} C_VEL
LIN {X 0,Y 587.365,Z 82.942,A -85,B 0,C 180,E1 -1606.153,E2 -1606.153} C_VEL
LIN {X 0,Y 587.348,Z 82.946,A -85,B 0,C 180,E1 -1608.961,E2 -1608.961} C_VEL
LIN {X 0,Y 587.347,Z 82.943,A -85,B 0,C 180,E1 -1611.742,E2 -1611.742} C_VEL
LIN {X 0,Y 587.349,Z 82.949,A -85,B 0,C 180,E1 -1614.505,E2 -1614.505} C_VEL
LIN {X 0,Y 587.371,Z 82.938,A -85,B 0,C 180,E1 -1617.255,E2 -1617.255} C_VEL
LIN {X 0,Y 587.39,Z 82.944,A -85,B 0,C 180,E1 -1619.998,E2 -1619.998} C_VEL
LIN {X 0,Y 587.361,Z 82.941,A -85,B 0,C 180,E1 -1622.741,E2 -1622.741} C_VEL
LIN {X 0,Y 587.36,Z 82.943,A -85,B 0,C 180,E1 -1625.49,E2 -1625.49} C_VEL
LIN {X 0,Y 587.34,Z 82.946,A -85,B 0,C 180,E1 -1628.253,E2 -1628.253} C_VEL
LIN {X 0,Y 587.351,Z 82.943,A -85,B 0,C 180,E1 -1631.131,E2 -1631.131} C_VEL
LIN {X 0,Y 587.331,Z 82.945,A -85,B 0,C 180,E1 -1634.244,E2 -1634.244} C_VEL
LIN {X 0,Y 587.336,Z 82.952,A -85,B 0,C 180,E1 -1637.403,E2 -1637.403} C_VEL
LIN {X 0,Y 587.293,Z 82.949,A -85,B 0,C 180,E1 -1638.281,E2 -1638.281} C_VEL
LIN {X 0,Y 586.656,Z 83.031,A -85,B 0,C 180,E1 -1638.853,E2 -1638.853} C_VEL
LIN {X 0,Y 583.847,Z 83.381,A -85,B 0,C 180,E1 -1639.782,E2 -1639.782} C_VEL
LIN {X 0,Y 581.441,Z 83.68,A -85,B 0,C 180,E1 -1640.529,E2 -1640.529} C_VEL
LIN {X 0,Y 580.38,Z 83.816,A -85,B 0,C 180,E1 -1641.105,E2 -1641.105} C_VEL
LIN {X 0,Y 580.279,Z 83.832,A -85,B 0,C 180,E1 -1641.301,E2 -1641.301} C_VEL
LIN {X 0,Y 580.257,Z 83.83,A -85,B 0,C 180,E1 -1643.556,E2 -1643.556} C_VEL
LIN {X 0,Y 580.28,Z 83.822,A -85,B 0,C 180,E1 -1646.33,E2 -1646.33} C_VEL
LIN {X 0,Y 580.284,Z 83.825,A -85,B 0,C 180,E1 -1649.305,E2 -1649.305} C_VEL
LIN {X 0,Y 580.284,Z 83.823,A -85,B 0,C 180,E1 -1652.197,E2 -1652.197} C_VEL
LIN {X 0,Y 580.275,Z 83.83,A -85,B 0,C 180,E1 -1654.693,E2 -1654.693} C_VEL
LIN {X 0,Y 580.28,Z 83.824,A -85,B 0,C 180,E1 -1657.265,E2 -1657.265} C_VEL
LIN {X 0,Y 580.27,Z 83.829,A -85,B 0,C 180,E1 -1660.267,E2 -1660.267} C_VEL
LIN {X 0,Y 580.263,Z 83.832,A -85,B 0,C 180,E1 -1662.703,E2 -1662.703} C_VEL
LIN {X 0,Y 580.236,Z 83.829,A -85,B 0,C 180,E1 -1665.607,E2 -1665.607} C_VEL
LIN {X 0,Y 580.249,Z 83.837,A -85,B 0,C 180,E1 -1668.227,E2 -1668.227} C_VEL
LIN {X 0,Y 580.246,Z 83.83,A -85,B 0,C 180,E1 -1670.961,E2 -1670.961} C_VEL
LIN {X 0,Y 580.296,Z 83.945,A -85,B 0,C 180,E1 -1672.776,E2 -1672.776} C_VEL
LIN {X 0,Y 580.724,Z 89.285,A -85,B 0,C 180,E1 -1673.629,E2 -1673.629} C_VEL
LIN {X 0,Y 580.55,Z 107.701,A -85,B 0,C 180,E1 -1676.439,E2 -1676.439} C_VEL
LIN {X 0,Y 580.476,Z 114.746,A -85,B 0,C 180,E1 -1677.5,E2 -1677.5} C_VEL
LIN {X 0,Y 581.402,Z 120.876,A -85,B 0,C 180,E1 -1677.606,E2 -1677.606} C_VEL
LIN {X 0,Y 581.15,Z 251.31,A -85,B 0,C 180,E1 -1679.255,E2 -1679.255} C_VEL
LIN {X 0,Y 581.053,Z 265.34,A -85,B 0,C 180,E1 -1679.569,E2 -1679.569} C_VEL
LIN {X 0,Y 580.944,Z 278.951,A -85,B 0,C 180,E1 -1680.014,E2 -1680.014} C_VEL
LIN {X 0,Y 580.824,Z 292.175,A -85,B 0,C 180,E1 -1680.591,E2 -1680.591} C_VEL
LIN {X 0,Y 580.669,Z 305.585,A -85,B 0,C 180,E1 -1681.34,E2 -1681.34} C_VEL
LIN {X 0,Y 580.546,Z 317.465,A -85,B 0,C 180,E1 -1682.167,E2 -1682.167} C_VEL
LIN {X 0,Y 580.437,Z 328.387,A -85,B 0,C 180,E1 -1683.092,E2 -1683.092} C_VEL
LIN {X 0,Y 580.293,Z 338.722,A -85,B 0,C 180,E1 -1684.15,E2 -1684.15} C_VEL
LIN {X 0,Y 580.231,Z 347.77,A -85,B 0,C 180,E1 -1685.28,E2 -1685.28} C_VEL
LIN {X 0,Y 580.174,Z 355.4,A -85,B 0,C 180,E1 -1686.437,E2 -1686.437} C_VEL
LIN {X 0,Y 580.118,Z 361.509,A -85,B 0,C 180,E1 -1687.565,E2 -1687.565} C_VEL
LIN {X 0,Y 580.096,Z 367.116,A -85,B 0,C 180,E1 -1688.875,E2 -1688.875} C_VEL
LIN {X 0,Y 580.077,Z 371.286,A -85,B 0,C 180,E1 -1690.169,E2 -1690.169} C_VEL
LIN {X 0,Y 580.026,Z 374.484,A -85,B 0,C 180,E1 -1691.636,E2 -1691.636} C_VEL
LIN {X 0,Y 580.04,Z 376.161,A -85,B 0,C 180,E1 -1693.094,E2 -1693.094} C_VEL
LIN {X 0,Y 580.048,Z 376.394,A -85,B 0,C 180,E1 -1694.54,E2 -1694.54} C_VEL
LIN {X 0,Y 580.092,Z 375.215,A -85,B 0,C 180,E1 -1695.976,E2 -1695.976} C_VEL
LIN {X 0,Y 580.067,Z 372.61,A -85,B 0,C 180,E1 -1697.402,E2 -1697.402} C_VEL
LIN {X 0,Y 580.095,Z 368.513,A -85,B 0,C 180,E1 -1698.822,E2 -1698.822} C_VEL
LIN {X 0,Y 580.105,Z 362.855,A -85,B 0,C 180,E1 -1700.234,E2 -1700.234} C_VEL
LIN {X 0,Y 580.158,Z 356.488,A -85,B 0,C 180,E1 -1701.465,E2 -1701.465} C_VEL
LIN {X 0,Y 580.195,Z 348.61,A -85,B 0,C 180,E1 -1702.692,E2 -1702.692} C_VEL
LIN {X 0,Y 580.275,Z 340.411,A -85,B 0,C 180,E1 -1703.741,E2 -1703.741} C_VEL
LIN {X 0,Y 580.401,Z 330.584,A -85,B 0,C 180,E1 -1704.788,E2 -1704.788} C_VEL
LIN {X 0,Y 580.516,Z 319.73,A -85,B 0,C 180,E1 -1705.747,E2 -1705.747} C_VEL
LIN {X 0,Y 580.643,Z 307.713,A -85,B 0,C 180,E1 -1706.616,E2 -1706.616} C_VEL
LIN {X 0,Y 580.768,Z 295.908,A -85,B 0,C 180,E1 -1707.311,E2 -1707.311} C_VEL
LIN {X 0,Y 580.903,Z 282.955,A -85,B 0,C 180,E1 -1707.919,E2 -1707.919} C_VEL
LIN {X 0,Y 581.022,Z 268.897,A -85,B 0,C 180,E1 -1708.418,E2 -1708.418} C_VEL
LIN {X 0,Y 581.091,Z 254.99,A -85,B 0,C 180,E1 -1708.765,E2 -1708.765} C_VEL
LIN {X 0,Y 581.136,Z 237.575,A -85,B 0,C 180,E1 -1709.025,E2 -1709.025} C_VEL
LIN {X 0,Y 581.312,Z 119.24,A -85,B 0,C 180,E1 -1710.508,E2 -1710.508} C_VEL
LIN {X 0,Y 580.467,Z 114.643,A -85,B 0,C 180,E1 -1710.606,E2 -1710.606} C_VEL
LIN {X 0,Y 580.656,Z 95.728,A -85,B 0,C 180,E1 -1713.469,E2 -1713.469} C_VEL
LIN {X 0,Y 580.622,Z 85.638,A -85,B 0,C 180,E1 -1715.033,E2 -1715.033} C_VEL
LIN {X 0,Y 580.328,Z 83.824,A -85,B 0,C 180,E1 -1715.341,E2 -1715.341} C_VEL
LIN {X 0,Y 580.331,Z 83.824,A -85,B 0,C 180,E1 -1717.654,E2 -1717.654} C_VEL
LIN {X 0,Y 580.292,Z 83.823,A -85,B 0,C 180,E1 -1720.466,E2 -1720.466} C_VEL
LIN {X 0,Y 580.281,Z 83.827,A -85,B 0,C 180,E1 -1723.303,E2 -1723.303} C_VEL
LIN {X 0,Y 580.296,Z 83.827,A -85,B 0,C 180,E1 -1725.452,E2 -1725.452} C_VEL
LIN {X 0,Y 580.282,Z 83.832,A -85,B 0,C 180,E1 -1727.624,E2 -1727.624} C_VEL
LIN {X 0,Y 580.286,Z 83.827,A -85,B 0,C 180,E1 -1729.822,E2 -1729.822} C_VEL
LIN {X 0,Y 580.318,Z 83.819,A -85,B 0,C 180,E1 -1732.8,E2 -1732.8} C_VEL
LIN {X 0,Y 580.274,Z 83.826,A -85,B 0,C 180,E1 -1735.849,E2 -1735.849} C_VEL
LIN {X 0,Y 580.281,Z 83.822,A -85,B 0,C 180,E1 -1738.185,E2 -1738.185} C_VEL
LIN {X 0,Y 580.278,Z 83.825,A -85,B 0,C 180,E1 -1740.701,E2 -1740.701} C_VEL
LIN {X 0,Y 580.301,Z 83.826,A -85,B 0,C 180,E1 -1743.323,E2 -1743.323} C_VEL
LIN {X 0,Y 580.302,Z 83.82,A -85,B 0,C 180,E1 -1745.771,E2 -1745.771} C_VEL
LIN {X 0,Y 580.28,Z 83.823,A -85,B 0,C 180,E1 -1748.145,E2 -1748.145} C_VEL
LIN {X 0,Y 580.297,Z 83.83,A -85,B 0,C 180,E1 -1750.842,E2 -1750.842} C_VEL
LIN {X 0,Y 580.26,Z 83.825,A -85,B 0,C 180,E1 -1753.658,E2 -1753.658} C_VEL
LIN {X 0,Y 580.269,Z 83.832,A -85,B 0,C 180,E1 -1756.608,E2 -1756.608} C_VEL
LIN {X 0,Y 580.295,Z 83.823,A -85,B 0,C 180,E1 -1759.161,E2 -1759.161} C_VEL
LIN {X 0,Y 580.267,Z 83.825,A -85,B 0,C 180,E1 -1761.928,E2 -1761.928} C_VEL
LIN {X 0,Y 580.286,Z 83.832,A -85,B 0,C 180,E1 -1764.459,E2 -1764.459} C_VEL
LIN {X 0,Y 580.276,Z 83.824,A -85,B 0,C 180,E1 -1766.978,E2 -1766.978} C_VEL
LIN {X 0,Y 580.288,Z 83.821,A -85,B 0,C 180,E1 -1769.428,E2 -1769.428} C_VEL
LIN {X 0,Y 580.298,Z 83.829,A -85,B 0,C 180,E1 -1772.139,E2 -1772.139} C_VEL
LIN {X 0,Y 580.292,Z 83.821,A -85,B 0,C 180,E1 -1774.923,E2 -1774.923} C_VEL
LIN {X 0,Y 580.331,Z 83.816,A -85,B 0,C 180,E1 -1777.202,E2 -1777.202} C_VEL
LIN {X 0,Y 580.293,Z 83.827,A -85,B 0,C 180,E1 -1780.18,E2 -1780.18} C_VEL
LIN {X 0,Y 580.312,Z 83.819,A -85,B 0,C 180,E1 -1783.106,E2 -1783.106} C_VEL
LIN {X 0,Y 580.312,Z 83.825,A -85,B 0,C 180,E1 -1785.986,E2 -1785.986} C_VEL
LIN {X 0,Y 580.316,Z 83.818,A -85,B 0,C 180,E1 -1788.83,E2 -1788.83} C_VEL
LIN {X 0,Y 580.325,Z 83.826,A -85,B 0,C 180,E1 -1791.646,E2 -1791.646} C_VEL
LIN {X 0,Y 580.32,Z 83.817,A -85,B 0,C 180,E1 -1794.443,E2 -1794.443} C_VEL
LIN {X 0,Y 580.341,Z 83.821,A -85,B 0,C 180,E1 -1797.226,E2 -1797.226} C_VEL
LIN {X 0,Y 580.339,Z 83.816,A -85,B 0,C 180,E1 -1800.002,E2 -1800.002} C_VEL
LIN {X 0,Y 580.339,Z 83.818,A -85,B 0,C 180,E1 -1802.779,E2 -1802.779} C_VEL
LIN {X 0,Y 580.319,Z 83.821,A -85,B 0,C 180,E1 -1805.562,E2 -1805.562} C_VEL
LIN {X 0,Y 580.326,Z 83.817,A -85,B 0,C 180,E1 -1808.358,E2 -1808.358} C_VEL
LIN {X 0,Y 580.292,Z 83.827,A -85,B 0,C 180,E1 -1811.193,E2 -1811.193} C_VEL
LIN {X 0,Y 580.319,Z 83.817,A -85,B 0,C 180,E1 -1814.019,E2 -1814.019} C_VEL
LIN {X 0,Y 580.306,Z 83.828,A -85,B 0,C 180,E1 -1816.916,E2 -1816.916} C_VEL
LIN {X 0,Y 580.301,Z 83.82,A -85,B 0,C 180,E1 -1819.824,E2 -1819.824} C_VEL
LIN {X 0,Y 580.29,Z 83.828,A -85,B 0,C 180,E1 -1822.804,E2 -1822.804} C_VEL
LIN {X 0,Y 580.303,Z 83.822,A -85,B 0,C 180,E1 -1825.081,E2 -1825.081} C_VEL
LIN {X 0,Y 580.316,Z 83.819,A -85,B 0,C 180,E1 -1827.865,E2 -1827.865} C_VEL
LIN {X 0,Y 580.279,Z 83.827,A -85,B 0,C 180,E1 -1830.696,E2 -1830.696} C_VEL
LIN {X 0,Y 580.302,Z 83.819,A -85,B 0,C 180,E1 -1833.318,E2 -1833.318} C_VEL
LIN {X 0,Y 580.272,Z 83.826,A -85,B 0,C 180,E1 -1835.762,E2 -1835.762} C_VEL
LIN {X 0,Y 580.286,Z 83.831,A -85,B 0,C 180,E1 -1838.148,E2 -1838.148} C_VEL
LIN {X 0,Y 580.296,Z 83.821,A -85,B 0,C 180,E1 -1840.845,E2 -1840.845} C_VEL
LIN {X 0,Y 580.286,Z 83.826,A -85,B 0,C 180,E1 -1843.658,E2 -1843.658} C_VEL
LIN {X 0,Y 580.274,Z 83.824,A -85,B 0,C 180,E1 -1846.611,E2 -1846.611} C_VEL
LIN {X 0,Y 580.296,Z 83.821,A -85,B 0,C 180,E1 -1849.158,E2 -1849.158} C_VEL
LIN {X 0,Y 580.289,Z 83.828,A -85,B 0,C 180,E1 -1851.928,E2 -1851.928} C_VEL
LIN {X 0,Y 580.25,Z 83.826,A -85,B 0,C 180,E1 -1854.454,E2 -1854.454} C_VEL
LIN {X 0,Y 580.288,Z 83.823,A -85,B 0,C 180,E1 -1856.976,E2 -1856.976} C_VEL
LIN {X 0,Y 580.286,Z 83.831,A -85,B 0,C 180,E1 -1859.426,E2 -1859.426} C_VEL
LIN {X 0,Y 580.297,Z 83.822,A -85,B 0,C 180,E1 -1862.143,E2 -1862.143} C_VEL
LIN {X 0,Y 580.32,Z 83.827,A -85,B 0,C 180,E1 -1865.271,E2 -1865.271} C_VEL
LIN {X 0,Y 580.324,Z 83.956,A -85,B 0,C 180,E1 -1865.655,E2 -1865.655} C_VEL
LIN {X 0,Y 581.078,Z 88.501,A -85,B 0,C 180,E1 -1866.289,E2 -1866.289} C_VEL
LIN {X 0,Y 580.928,Z 109.916,A -85,B 0,C 180,E1 -1869.092,E2 -1869.092} C_VEL
LIN {X 0,Y 580.739,Z 131.13,A -85,B 0,C 180,E1 -1871.844,E2 -1871.844} C_VEL
LIN {X 0,Y 580.593,Z 143.582,A -85,B 0,C 180,E1 -1873.44,E2 -1873.44} C_VEL
LIN {X 0,Y 581.41,Z 149.493,A -85,B 0,C 180,E1 -1873.543,E2 -1873.543} C_VEL
LIN {X 0,Y 581.121,Z 281.941,A -85,B 0,C 180,E1 -1875.221,E2 -1875.221} C_VEL
LIN {X 0,Y 581.042,Z 296.51,A -85,B 0,C 180,E1 -1875.558,E2 -1875.558} C_VEL
LIN {X 0,Y 580.911,Z 310.866,A -85,B 0,C 180,E1 -1876.043,E2 -1876.043} C_VEL
LIN {X 0,Y 580.805,Z 323.665,A -85,B 0,C 180,E1 -1876.62,E2 -1876.62} C_VEL
LIN {X 0,Y 580.655,Z 336.119,A -85,B 0,C 180,E1 -1877.329,E2 -1877.329} C_VEL
LIN {X 0,Y 580.524,Z 348.657,A -85,B 0,C 180,E1 -1878.213,E2 -1878.213} C_VEL
LIN {X 0,Y 580.44,Z 359.903,A -85,B 0,C 180,E1 -1879.19,E2 -1879.19} C_VEL
LIN {X 0,Y 580.275,Z 369.86,A -85,B 0,C 180,E1 -1880.239,E2 -1880.239} C_VEL
LIN {X 0,Y 580.241,Z 378.18,A -85,B 0,C 180,E1 -1881.293,E2 -1881.293} C_VEL
LIN {X 0,Y 580.166,Z 386.133,A -85,B 0,C 180,E1 -1882.519,E2 -1882.519} C_VEL
LIN {X 0,Y 580.103,Z 392.532,A -85,B 0,C 180,E1 -1883.741,E2 -1883.741} C_VEL
LIN {X 0,Y 580.077,Z 396.965,A -85,B 0,C 180,E1 -1884.788,E2 -1884.788} C_VEL
LIN {X 0,Y 580.103,Z 400.446,A -85,B 0,C 180,E1 -1885.832,E2 -1885.832} C_VEL
LIN {X 0,Y 580.04,Z 403.834,A -85,B 0,C 180,E1 -1887.223,E2 -1887.223} C_VEL
LIN {X 0,Y 580.042,Z 405.834,A -85,B 0,C 180,E1 -1888.612,E2 -1888.612} C_VEL
LIN {X 0,Y 580.036,Z 406.5,A -85,B 0,C 180,E1 -1890.001,E2 -1890.001} C_VEL
LIN {X 0,Y 580.042,Z 405.832,A -85,B 0,C 180,E1 -1891.39,E2 -1891.39} C_VEL
LIN {X 0,Y 580.04,Z 403.832,A -85,B 0,C 180,E1 -1892.779,E2 -1892.779} C_VEL
LIN {X 0,Y 580.104,Z 400.442,A -85,B 0,C 180,E1 -1894.169,E2 -1894.169} C_VEL
LIN {X 0,Y 580.129,Z 395.564,A -85,B 0,C 180,E1 -1895.563,E2 -1895.563} C_VEL
LIN {X 0,Y 580.143,Z 389.048,A -85,B 0,C 180,E1 -1896.959,E2 -1896.959} C_VEL
LIN {X 0,Y 580.193,Z 381.795,A -85,B 0,C 180,E1 -1898.184,E2 -1898.184} C_VEL
LIN {X 0,Y 580.284,Z 372.814,A -85,B 0,C 180,E1 -1899.411,E2 -1899.411} C_VEL
LIN {X 0,Y 580.357,Z 363.382,A -85,B 0,C 180,E1 -1900.467,E2 -1900.467} C_VEL
LIN {X 0,Y 580.472,Z 353.31,A -85,B 0,C 180,E1 -1901.405,E2 -1901.405} C_VEL
LIN {X 0,Y 580.597,Z 341.421,A -85,B 0,C 180,E1 -1902.319,E2 -1902.319} C_VEL
LIN {X 0,Y 580.725,Z 328.627,A -85,B 0,C 180,E1 -1903.116,E2 -1903.116} C_VEL
LIN {X 0,Y 580.886,Z 316.132,A -85,B 0,C 180,E1 -1903.736,E2 -1903.736} C_VEL
LIN {X 0,Y 581.005,Z 303.22,A -85,B 0,C 180,E1 -1904.235,E2 -1904.235} C_VEL
LIN {X 0,Y 581.087,Z 289.156,A -85,B 0,C 180,E1 -1904.631,E2 -1904.631} C_VEL
LIN {X 0,Y 581.163,Z 274.533,A -85,B 0,C 180,E1 -1904.892,E2 -1904.892} C_VEL
LIN {X 0,Y 581.35,Z 147.767,A -85,B 0,C 180,E1 -1906.48,E2 -1906.48} C_VEL
LIN {X 0,Y 580.596,Z 143.478,A -85,B 0,C 180,E1 -1906.573,E2 -1906.573} C_VEL
LIN {X 0,Y 580.791,Z 122.365,A -85,B 0,C 180,E1 -1909.289,E2 -1909.289} C_VEL
LIN {X 0,Y 580.989,Z 101.317,A -85,B 0,C 180,E1 -1912.025,E2 -1912.025} C_VEL
LIN {X 0,Y 581.081,Z 88.438,A -85,B 0,C 180,E1 -1913.713,E2 -1913.713} C_VEL
LIN {X 0,Y 580.312,Z 83.828,A -85,B 0,C 180,E1 -1914.379,E2 -1914.379} C_VEL
LIN {X 0,Y 580.289,Z 83.823,A -85,B 0,C 180,E1 -1917.403,E2 -1917.403} C_VEL
LIN {X 0,Y 580.285,Z 83.824,A -85,B 0,C 180,E1 -1919.774,E2 -1919.774} C_VEL
LIN {X 0,Y 580.306,Z 83.828,A -85,B 0,C 180,E1 -1922.201,E2 -1922.201} C_VEL
LIN {X 0,Y 580.295,Z 83.825,A -85,B 0,C 180,E1 -1924.697,E2 -1924.697} C_VEL
LIN {X 0,Y 580.298,Z 83.82,A -85,B 0,C 180,E1 -1927.269,E2 -1927.269} C_VEL
LIN {X 0,Y 580.298,Z 83.826,A -85,B 0,C 180,E1 -1930.27,E2 -1930.27} C_VEL
LIN {X 0,Y 580.282,Z 83.823,A -85,B 0,C 180,E1 -1932.707,E2 -1932.707} C_VEL
LIN {X 0,Y 580.266,Z 83.83,A -85,B 0,C 180,E1 -1935.611,E2 -1935.611} C_VEL
LIN {X 0,Y 580.289,Z 83.822,A -85,B 0,C 180,E1 -1938.231,E2 -1938.231} C_VEL
LIN {X 0,Y 580.279,Z 83.824,A -85,B 0,C 180,E1 -1940.964,E2 -1940.964} C_VEL
LIN {X 0,Y 580.26,Z 83.834,A -85,B 0,C 180,E1 -1943.594,E2 -1943.594} C_VEL
LIN {X 0,Y 580.291,Z 83.822,A -85,B 0,C 180,E1 -1946.142,E2 -1946.142} C_VEL
LIN {X 0,Y 580.281,Z 83.823,A -85,B 0,C 180,E1 -1948.613,E2 -1948.613} C_VEL
LIN {X 0,Y 580.299,Z 83.826,A -85,B 0,C 180,E1 -1951.023,E2 -1951.023} C_VEL
LIN {X 0,Y 580.28,Z 83.825,A -85,B 0,C 180,E1 -1953.67,E2 -1953.67} C_VEL
LIN {X 0,Y 580.303,Z 83.82,A -85,B 0,C 180,E1 -1955.682,E2 -1955.682} C_VEL
LIN {X 0,Y 580.295,Z 83.826,A -85,B 0,C 180,E1 -1958.693,E2 -1958.693} C_VEL
LIN {X 0,Y 580.303,Z 83.829,A -85,B 0,C 180,E1 -1960.912,E2 -1960.912} C_VEL
LIN {X 0,Y 580.273,Z 83.823,A -85,B 0,C 180,E1 -1963.824,E2 -1963.824} C_VEL
LIN {X 0,Y 580.324,Z 83.818,A -85,B 0,C 180,E1 -1965.981,E2 -1965.981} C_VEL
LIN {X 0,Y 580.316,Z 83.824,A -85,B 0,C 180,E1 -1968.825,E2 -1968.825} C_VEL
LIN {X 0,Y 580.316,Z 83.818,A -85,B 0,C 180,E1 -1971.642,E2 -1971.642} C_VEL
LIN {X 0,Y 580.316,Z 83.827,A -85,B 0,C 180,E1 -1974.438,E2 -1974.438} C_VEL
LIN {X 0,Y 580.338,Z 83.814,A -85,B 0,C 180,E1 -1977.221,E2 -1977.221} C_VEL
LIN {X 0,Y 580.359,Z 83.82,A -85,B 0,C 180,E1 -1979.998,E2 -1979.998} C_VEL
LIN {X 0,Y 580.329,Z 83.817,A -85,B 0,C 180,E1 -1982.774,E2 -1982.774} C_VEL
LIN {X 0,Y 580.325,Z 83.82,A -85,B 0,C 180,E1 -1985.557,E2 -1985.557} C_VEL
LIN {X 0,Y 580.31,Z 83.821,A -85,B 0,C 180,E1 -1988.354,E2 -1988.354} C_VEL
LIN {X 0,Y 580.303,Z 83.822,A -85,B 0,C 180,E1 -1991.188,E2 -1991.188} C_VEL
LIN {X 0,Y 580.306,Z 83.823,A -85,B 0,C 180,E1 -1994.015,E2 -1994.015} C_VEL
LIN {X 0,Y 580.288,Z 83.823,A -85,B 0,C 180,E1 -1996.903,E2 -1996.903} C_VEL
LIN {X 0,Y 580.278,Z 83.825,A -85,B 0,C 180,E1 -1999.82,E2 -1999.82} C_VEL
LIN {X 0,Y 580.279,Z 83.832,A -85,B 0,C 180,E1 -2001.301,E2 -2001.301} C_VEL
LIN {X 0,Y 579.57,Z 83.927,A -85,B 0,C 180,E1 -2001.88,E2 -2001.88} C_VEL
LIN {X 0,Y 576.69,Z 84.282,A -85,B 0,C 180,E1 -2002.82,E2 -2002.82} C_VEL
LIN {X 0,Y 574.293,Z 84.573,A -85,B 0,C 180,E1 -2003.576,E2 -2003.576} C_VEL
LIN {X 0,Y 573.283,Z 84.694,A -85,B 0,C 180,E1 -2004.16,E2 -2004.16} C_VEL
LIN {X 0,Y 573.21,Z 84.704,A -85,B 0,C 180,E1 -2004.357,E2 -2004.357} C_VEL
LIN {X 0,Y 573.239,Z 84.707,A -85,B 0,C 180,E1 -2006.973,E2 -2006.973} C_VEL
LIN {X 0,Y 573.228,Z 84.702,A -85,B 0,C 180,E1 -2009.483,E2 -2009.483} C_VEL
LIN {X 0,Y 573.239,Z 84.706,A -85,B 0,C 180,E1 -2012.642,E2 -2012.642} C_VEL
LIN {X 0,Y 573.193,Z 84.71,A -85,B 0,C 180,E1 -2015.185,E2 -2015.185} C_VEL
LIN {X 0,Y 573.215,Z 84.702,A -85,B 0,C 180,E1 -2017.805,E2 -2017.805} C_VEL
LIN {X 0,Y 573.227,Z 84.71,A -85,B 0,C 180,E1 -2020.522,E2 -2020.522} C_VEL
LIN {X 0,Y 573.217,Z 84.703,A -85,B 0,C 180,E1 -2023.356,E2 -2023.356} C_VEL
LIN {X 0,Y 573.212,Z 84.713,A -85,B 0,C 180,E1 -2026.329,E2 -2026.329} C_VEL
LIN {X 0,Y 573.2,Z 84.713,A -85,B 0,C 180,E1 -2028.539,E2 -2028.539} C_VEL
LIN {X 0,Y 573.212,Z 84.707,A -85,B 0,C 180,E1 -2031.295,E2 -2031.295} C_VEL
LIN {X 0,Y 573.264,Z 84.868,A -85,B 0,C 180,E1 -2032.622,E2 -2032.622} C_VEL
LIN {X 0,Y 573.832,Z 89.247,A -85,B 0,C 180,E1 -2033.339,E2 -2033.339} C_VEL
LIN {X 0,Y 573.577,Z 108.228,A -85,B 0,C 180,E1 -2036.299,E2 -2036.299} C_VEL
LIN {X 0,Y 573.527,Z 114.85,A -85,B 0,C 180,E1 -2037.296,E2 -2037.296} C_VEL
LIN {X 0,Y 574.597,Z 121.554,A -85,B 0,C 180,E1 -2037.414,E2 -2037.414} C_VEL
LIN {X 0,Y 574.304,Z 251.074,A -85,B 0,C 180,E1 -2039.07,E2 -2039.07} C_VEL
LIN {X 0,Y 574.168,Z 265.42,A -85,B 0,C 180,E1 -2039.394,E2 -2039.394} C_VEL
LIN {X 0,Y 574.059,Z 278.387,A -85,B 0,C 180,E1 -2039.819,E2 -2039.819} C_VEL
LIN {X 0,Y 573.907,Z 291.429,A -85,B 0,C 180,E1 -2040.387,E2 -2040.387} C_VEL
LIN {X 0,Y 573.73,Z 303.636,A -85,B 0,C 180,E1 -2041.061,E2 -2041.061} C_VEL
LIN {X 0,Y 573.568,Z 315.929,A -85,B 0,C 180,E1 -2041.903,E2 -2041.903} C_VEL
LIN {X 0,Y 573.433,Z 327.067,A -85,B 0,C 180,E1 -2042.835,E2 -2042.835} C_VEL
LIN {X 0,Y 573.308,Z 336.754,A -85,B 0,C 180,E1 -2043.811,E2 -2043.811} C_VEL
LIN {X 0,Y 573.182,Z 345.71,A -85,B 0,C 180,E1 -2044.893,E2 -2044.893} C_VEL
LIN {X 0,Y 573.097,Z 354.115,A -85,B 0,C 180,E1 -2046.128,E2 -2046.128} C_VEL
LIN {X 0,Y 573.058,Z 360.45,A -85,B 0,C 180,E1 -2047.274,E2 -2047.274} C_VEL
LIN {X 0,Y 573.038,Z 365.554,A -85,B 0,C 180,E1 -2048.411,E2 -2048.411} C_VEL
LIN {X 0,Y 572.991,Z 369.582,A -85,B 0,C 180,E1 -2049.538,E2 -2049.538} C_VEL
LIN {X 0,Y 572.958,Z 372.963,A -85,B 0,C 180,E1 -2050.808,E2 -2050.808} C_VEL
LIN {X 0,Y 572.93,Z 375.274,A -85,B 0,C 180,E1 -2052.14,E2 -2052.14} C_VEL
LIN {X 0,Y 572.937,Z 376.409,A -85,B 0,C 180,E1 -2053.612,E2 -2053.612} C_VEL
LIN {X 0,Y 572.956,Z 376.118,A -85,B 0,C 180,E1 -2055.072,E2 -2055.072} C_VEL
LIN {X 0,Y 572.987,Z 374.418,A -85,B 0,C 180,E1 -2056.523,E2 -2056.523} C_VEL
LIN {X 0,Y 572.996,Z 371.297,A -85,B 0,C 180,E1 -2057.964,E2 -2057.964} C_VEL
LIN {X 0,Y 573.025,Z 366.685,A -85,B 0,C 180,E1 -2059.398,E2 -2059.398} C_VEL
LIN {X 0,Y 573.027,Z 362.134,A -85,B 0,C 180,E1 -2060.469,E2 -2060.469} C_VEL
LIN {X 0,Y 573.085,Z 355.593,A -85,B 0,C 180,E1 -2061.714,E2 -2061.714} C_VEL
LIN {X 0,Y 573.181,Z 347.514,A -85,B 0,C 180,E1 -2062.956,E2 -2062.956} C_VEL
LIN {X 0,Y 573.284,Z 337.526,A -85,B 0,C 180,E1 -2064.194,E2 -2064.194} C_VEL
LIN {X 0,Y 573.4,Z 327.089,A -85,B 0,C 180,E1 -2065.253,E2 -2065.253} C_VEL
LIN {X 0,Y 573.539,Z 315.47,A -85,B 0,C 180,E1 -2066.223,E2 -2066.223} C_VEL
LIN {X 0,Y 573.703,Z 303.868,A -85,B 0,C 180,E1 -2067.015,E2 -2067.015} C_VEL
LIN {X 0,Y 573.888,Z 291.138,A -85,B 0,C 180,E1 -2067.718,E2 -2067.718} C_VEL
LIN {X 0,Y 574.076,Z 277.926,A -85,B 0,C 180,E1 -2068.289,E2 -2068.289} C_VEL
LIN {X 0,Y 574.163,Z 263.479,A -85,B 0,C 180,E1 -2068.75,E2 -2068.75} C_VEL
LIN {X 0,Y 574.244,Z 248.77,A -85,B 0,C 180,E1 -2069.057,E2 -2069.057} C_VEL
LIN {X 0,Y 574.467,Z 119.99,A -85,B 0,C 180,E1 -2070.7,E2 -2070.7} C_VEL
LIN {X 0,Y 573.484,Z 114.66,A -85,B 0,C 180,E1 -2070.811,E2 -2070.811} C_VEL
LIN {X 0,Y 573.707,Z 96.025,A -85,B 0,C 180,E1 -2073.686,E2 -2073.686} C_VEL
LIN {X 0,Y 573.693,Z 87.086,A -85,B 0,C 180,E1 -2075.094,E2 -2075.094} C_VEL
LIN {X 0,Y 573.279,Z 84.703,A -85,B 0,C 180,E1 -2075.495,E2 -2075.495} C_VEL
LIN {X 0,Y 573.279,Z 84.703,A -85,B 0,C 180,E1 -2077.749,E2 -2077.749} C_VEL
LIN {X 0,Y 573.259,Z 84.699,A -85,B 0,C 180,E1 -2080.596,E2 -2080.596} C_VEL
LIN {X 0,Y 573.237,Z 84.707,A -85,B 0,C 180,E1 -2083.469,E2 -2083.469} C_VEL
LIN {X 0,Y 573.257,Z 84.707,A -85,B 0,C 180,E1 -2085.646,E2 -2085.646} C_VEL
LIN {X 0,Y 573.234,Z 84.706,A -85,B 0,C 180,E1 -2087.848,E2 -2087.848} C_VEL
LIN {X 0,Y 573.234,Z 84.701,A -85,B 0,C 180,E1 -2090.826,E2 -2090.826} C_VEL
LIN {X 0,Y 573.27,Z 84.701,A -85,B 0,C 180,E1 -2093.163,E2 -2093.163} C_VEL
LIN {X 0,Y 573.262,Z 84.697,A -85,B 0,C 180,E1 -2096.189,E2 -2096.189} C_VEL
LIN {X 0,Y 573.24,Z 84.7,A -85,B 0,C 180,E1 -2098.563,E2 -2098.563} C_VEL
LIN {X 0,Y 573.22,Z 84.708,A -85,B 0,C 180,E1 -2100.992,E2 -2100.992} C_VEL
LIN {X 0,Y 573.251,Z 84.701,A -85,B 0,C 180,E1 -2103.529,E2 -2103.529} C_VEL
LIN {X 0,Y 573.261,Z 84.697,A -85,B 0,C 180,E1 -2106.047,E2 -2106.047} C_VEL
LIN {X 0,Y 573.234,Z 84.706,A -85,B 0,C 180,E1 -2108.701,E2 -2108.701} C_VEL
LIN {X 0,Y 573.231,Z 84.702,A -85,B 0,C 180,E1 -2111.455,E2 -2111.455} C_VEL
LIN {X 0,Y 573.214,Z 84.706,A -85,B 0,C 180,E1 -2114.334,E2 -2114.334} C_VEL
LIN {X 0,Y 573.23,Z 84.71,A -85,B 0,C 180,E1 -2116.645,E2 -2116.645} C_VEL
LIN {X 0,Y 573.242,Z 84.699,A -85,B 0,C 180,E1 -2119.479,E2 -2119.479} C_VEL
LIN {X 0,Y 573.213,Z 84.707,A -85,B 0,C 180,E1 -2122.195,E2 -2122.195} C_VEL
LIN {X 0,Y 573.247,Z 84.702,A -85,B 0,C 180,E1 -2124.819,E2 -2124.819} C_VEL
LIN {X 0,Y 573.237,Z 84.7,A -85,B 0,C 180,E1 -2127.358,E2 -2127.358} C_VEL
LIN {X 0,Y 573.235,Z 84.703,A -85,B 0,C 180,E1 -2129.827,E2 -2129.827} C_VEL
LIN {X 0,Y 573.268,Z 84.705,A -85,B 0,C 180,E1 -2132.238,E2 -2132.238} C_VEL
LIN {X 0,Y 573.251,Z 84.698,A -85,B 0,C 180,E1 -2135.122,E2 -2135.122} C_VEL
LIN {X 0,Y 573.248,Z 84.702,A -85,B 0,C 180,E1 -2137.666,E2 -2137.666} C_VEL
LIN {X 0,Y 573.26,Z 84.697,A -85,B 0,C 180,E1 -2140.73,E2 -2140.73} C_VEL
LIN {X 0,Y 573.247,Z 84.704,A -85,B 0,C 180,E1 -2143.625,E2 -2143.625} C_VEL
LIN {X 0,Y 573.228,Z 84.701,A -85,B 0,C 180,E1 -2146.532,E2 -2146.532} C_VEL
LIN {X 0,Y 573.268,Z 84.696,A -85,B 0,C 180,E1 -2148.736,E2 -2148.736} C_VEL
LIN {X 0,Y 573.297,Z 84.701,A -85,B 0,C 180,E1 -2151.543,E2 -2151.543} C_VEL
LIN {X 0,Y 573.285,Z 84.694,A -85,B 0,C 180,E1 -2154.374,E2 -2154.374} C_VEL
LIN {X 0,Y 573.307,Z 84.697,A -85,B 0,C 180,E1 -2157.192,E2 -2157.192} C_VEL
LIN {X 0,Y 573.309,Z 84.692,A -85,B 0,C 180,E1 -2160.002,E2 -2160.002} C_VEL
LIN {X 0,Y 573.305,Z 84.694,A -85,B 0,C 180,E1 -2162.813,E2 -2162.813} C_VEL
LIN {X 0,Y 573.286,Z 84.697,A -85,B 0,C 180,E1 -2165.63,E2 -2165.63} C_VEL
LIN {X 0,Y 573.283,Z 84.695,A -85,B 0,C 180,E1 -2168.462,E2 -2168.462} C_VEL
LIN {X 0,Y 573.264,Z 84.701,A -85,B 0,C 180,E1 -2171.314,E2 -2171.314} C_VEL
LIN {X 0,Y 573.266,Z 84.697,A -85,B 0,C 180,E1 -2174.195,E2 -2174.195} C_VEL
LIN {X 0,Y 573.252,Z 84.703,A -85,B 0,C 180,E1 -2177.114,E2 -2177.114} C_VEL
LIN {X 0,Y 573.248,Z 84.699,A -85,B 0,C 180,E1 -2180.078,E2 -2180.078} C_VEL
LIN {X 0,Y 573.229,Z 84.703,A -85,B 0,C 180,E1 -2183.101,E2 -2183.101} C_VEL
LIN {X 0,Y 573.252,Z 84.698,A -85,B 0,C 180,E1 -2185.412,E2 -2185.412} C_VEL
LIN {X 0,Y 573.261,Z 84.7,A -85,B 0,C 180,E1 -2188.033,E2 -2188.033} C_VEL
LIN {X 0,Y 573.225,Z 84.704,A -85,B 0,C 180,E1 -2190.884,E2 -2190.884} C_VEL
LIN {X 0,Y 573.259,Z 84.697,A -85,B 0,C 180,E1 -2193.526,E2 -2193.526} C_VEL
LIN {X 0,Y 573.241,Z 84.706,A -85,B 0,C 180,E1 -2196.051,E2 -2196.051} C_VEL
LIN {X 0,Y 573.24,Z 84.701,A -85,B 0,C 180,E1 -2198.703,E2 -2198.703} C_VEL
LIN {X 0,Y 573.251,Z 84.701,A -85,B 0,C 180,E1 -2201.597,E2 -2201.597} C_VEL
LIN {X 0,Y 573.238,Z 84.704,A -85,B 0,C 180,E1 -2204.334,E2 -2204.334} C_VEL
LIN {X 0,Y 573.238,Z 84.702,A -85,B 0,C 180,E1 -2207.36,E2 -2207.36} C_VEL
LIN {X 0,Y 573.238,Z 84.701,A -85,B 0,C 180,E1 -2210.394,E2 -2210.394} C_VEL
LIN {X 0,Y 573.251,Z 84.699,A -85,B 0,C 180,E1 -2213.079,E2 -2213.079} C_VEL
LIN {X 0,Y 573.263,Z 84.706,A -85,B 0,C 180,E1 -2215.673,E2 -2215.673} C_VEL
LIN {X 0,Y 573.239,Z 84.701,A -85,B 0,C 180,E1 -2218.186,E2 -2218.186} C_VEL
LIN {X 0,Y 573.258,Z 84.699,A -85,B 0,C 180,E1 -2220.635,E2 -2220.635} C_VEL
LIN {X 0,Y 573.25,Z 84.704,A -85,B 0,C 180,E1 -2223.025,E2 -2223.025} C_VEL
LIN {X 0,Y 573.288,Z 84.756,A -85,B 0,C 180,E1 -2225.464,E2 -2225.464} C_VEL
LIN {X 0,Y 574.22,Z 90.831,A -85,B 0,C 180,E1 -2226.323,E2 -2226.323} C_VEL
LIN {X 0,Y 573.978,Z 112.616,A -85,B 0,C 180,E1 -2229.202,E2 -2229.202} C_VEL
LIN {X 0,Y 573.743,Z 133.956,A -85,B 0,C 180,E1 -2231.984,E2 -2231.984} C_VEL
LIN {X 0,Y 573.638,Z 143.597,A -85,B 0,C 180,E1 -2233.236,E2 -2233.236} C_VEL
LIN {X 0,Y 574.61,Z 149.613,A -85,B 0,C 180,E1 -2233.344,E2 -2233.344} C_VEL
LIN {X 0,Y 574.274,Z 281.941,A -85,B 0,C 180,E1 -2235.041,E2 -2235.041} C_VEL
LIN {X 0,Y 574.144,Z 296.509,A -85,B 0,C 180,E1 -2235.38,E2 -2235.38} C_VEL
LIN {X 0,Y 573.992,Z 310.864,A -85,B 0,C 180,E1 -2235.872,E2 -2235.872} C_VEL
LIN {X 0,Y 573.873,Z 323.662,A -85,B 0,C 180,E1 -2236.456,E2 -2236.456} C_VEL
LIN {X 0,Y 573.716,Z 336.12,A -85,B 0,C 180,E1 -2237.173,E2 -2237.173} C_VEL
LIN {X 0,Y 573.531,Z 348.66,A -85,B 0,C 180,E1 -2238.067,E2 -2238.067} C_VEL
LIN {X 0,Y 573.437,Z 360.153,A -85,B 0,C 180,E1 -2239.081,E2 -2239.081} C_VEL
LIN {X 0,Y 573.239,Z 369.861,A -85,B 0,C 180,E1 -2240.118,E2 -2240.118} C_VEL
LIN {X 0,Y 573.202,Z 378.181,A -85,B 0,C 180,E1 -2241.185,E2 -2241.185} C_VEL
LIN {X 0,Y 573.11,Z 386.134,A -85,B 0,C 180,E1 -2242.426,E2 -2242.426} C_VEL
LIN {X 0,Y 573.021,Z 392.533,A -85,B 0,C 180,E1 -2243.664,E2 -2243.664} C_VEL
LIN {X 0,Y 573,Z 396.965,A -85,B 0,C 180,E1 -2244.723,E2 -2244.723} C_VEL
LIN {X 0,Y 573.029,Z 400.446,A -85,B 0,C 180,E1 -2245.781,E2 -2245.781} C_VEL
LIN {X 0,Y 572.955,Z 403.834,A -85,B 0,C 180,E1 -2247.189,E2 -2247.189} C_VEL
LIN {X 0,Y 572.942,Z 405.834,A -85,B 0,C 180,E1 -2248.595,E2 -2248.595} C_VEL
LIN {X 0,Y 572.936,Z 406.5,A -85,B 0,C 180,E1 -2250.001,E2 -2250.001} C_VEL
LIN {X 0,Y 572.941,Z 405.833,A -85,B 0,C 180,E1 -2251.407,E2 -2251.407} C_VEL
LIN {X 0,Y 572.956,Z 403.832,A -85,B 0,C 180,E1 -2252.813,E2 -2252.813} C_VEL
LIN {X 0,Y 573.029,Z 400.443,A -85,B 0,C 180,E1 -2254.221,E2 -2254.221} C_VEL
LIN {X 0,Y 573.057,Z 395.564,A -85,B 0,C 180,E1 -2255.631,E2 -2255.631} C_VEL
LIN {X 0,Y 573.067,Z 390.819,A -85,B 0,C 180,E1 -2256.699,E2 -2256.699} C_VEL
LIN {X 0,Y 573.128,Z 384.03,A -85,B 0,C 180,E1 -2257.93,E2 -2257.93} C_VEL
LIN {X 0,Y 573.226,Z 375.55,A -85,B 0,C 180,E1 -2259.172,E2 -2259.172} C_VEL
LIN {X 0,Y 573.305,Z 366.698,A -85,B 0,C 180,E1 -2260.24,E2 -2260.24} C_VEL
LIN {X 0,Y 573.466,Z 355.978,A -85,B 0,C 180,E1 -2261.309,E2 -2261.309} C_VEL
LIN {X 0,Y 573.617,Z 345.125,A -85,B 0,C 180,E1 -2262.202,E2 -2262.202} C_VEL
LIN {X 0,Y 573.762,Z 333.239,A -85,B 0,C 180,E1 -2263.008,E2 -2263.008} C_VEL
LIN {X 0,Y 573.935,Z 320.076,A -85,B 0,C 180,E1 -2263.725,E2 -2263.725} C_VEL
LIN {X 0,Y 574.12,Z 306.806,A -85,B 0,C 180,E1 -2264.284,E2 -2264.284} C_VEL
LIN {X 0,Y 574.205,Z 292.797,A -85,B 0,C 180,E1 -2264.72,E2 -2264.72} C_VEL
LIN {X 0,Y 574.279,Z 279.066,A -85,B 0,C 180,E1 -2265.006,E2 -2265.006} C_VEL
LIN {X 0,Y 574.514,Z 148.56,A -85,B 0,C 180,E1 -2266.672,E2 -2266.672} C_VEL
LIN {X 0,Y 573.617,Z 143.505,A -85,B 0,C 180,E1 -2266.777,E2 -2266.777} C_VEL
LIN {X 0,Y 573.851,Z 123.059,A -85,B 0,C 180,E1 -2269.433,E2 -2269.433} C_VEL
LIN {X 0,Y 574.102,Z 101.133,A -85,B 0,C 180,E1 -2272.303,E2 -2272.303} C_VEL
LIN {X 0,Y 574.165,Z 89.703,A -85,B 0,C 180,E1 -2273.825,E2 -2273.825} C_VEL
LIN {X 0,Y 573.261,Z 84.707,A -85,B 0,C 180,E1 -2274.539,E2 -2274.539} C_VEL
LIN {X 0,Y 573.226,Z 84.706,A -85,B 0,C 180,E1 -2276.978,E2 -2276.978} C_VEL
LIN {X 0,Y 573.247,Z 84.7,A -85,B 0,C 180,E1 -2279.487,E2 -2279.487} C_VEL
LIN {X 0,Y 573.261,Z 84.704,A -85,B 0,C 180,E1 -2282.645,E2 -2282.645} C_VEL
LIN {X 0,Y 573.213,Z 84.704,A -85,B 0,C 180,E1 -2285.188,E2 -2285.188} C_VEL
LIN {X 0,Y 573.242,Z 84.703,A -85,B 0,C 180,E1 -2287.808,E2 -2287.808} C_VEL
LIN {X 0,Y 573.256,Z 84.7,A -85,B 0,C 180,E1 -2290.525,E2 -2290.525} C_VEL
LIN {X 0,Y 573.219,Z 84.704,A -85,B 0,C 180,E1 -2293.362,E2 -2293.362} C_VEL
LIN {X 0,Y 573.25,Z 84.701,A -85,B 0,C 180,E1 -2296.332,E2 -2296.332} C_VEL
LIN {X 0,Y 573.238,Z 84.697,A -85,B 0,C 180,E1 -2298.542,E2 -2298.542} C_VEL
LIN {X 0,Y 573.247,Z 84.703,A -85,B 0,C 180,E1 -2301.297,E2 -2301.297} C_VEL
LIN {X 0,Y 573.205,Z 84.707,A -85,B 0,C 180,E1 -2304.021,E2 -2304.021} C_VEL
LIN {X 0,Y 573.243,Z 84.699,A -85,B 0,C 180,E1 -2306.515,E2 -2306.515} C_VEL
LIN {X 0,Y 573.233,Z 84.706,A -85,B 0,C 180,E1 -2309.119,E2 -2309.119} C_VEL
LIN {X 0,Y 573.234,Z 84.7,A -85,B 0,C 180,E1 -2311.976,E2 -2311.976} C_VEL
LIN {X 0,Y 573.252,Z 84.7,A -85,B 0,C 180,E1 -2314.588,E2 -2314.588} C_VEL
LIN {X 0,Y 573.236,Z 84.701,A -85,B 0,C 180,E1 -2317.661,E2 -2317.661} C_VEL
LIN {X 0,Y 573.278,Z 84.7,A -85,B 0,C 180,E1 -2320.669,E2 -2320.669} C_VEL
LIN {X 0,Y 573.25,Z 84.698,A -85,B 0,C 180,E1 -2323.62,E2 -2323.62} C_VEL
LIN {X 0,Y 573.268,Z 84.696,A -85,B 0,C 180,E1 -2325.805,E2 -2325.805} C_VEL
LIN {X 0,Y 573.274,Z 84.702,A -85,B 0,C 180,E1 -2328.743,E2 -2328.743} C_VEL
LIN {X 0,Y 573.26,Z 84.697,A -85,B 0,C 180,E1 -2331.538,E2 -2331.538} C_VEL
LIN {X 0,Y 573.283,Z 84.704,A -85,B 0,C 180,E1 -2334.37,E2 -2334.37} C_VEL
LIN {X 0,Y 573.314,Z 84.694,A -85,B 0,C 180,E1 -2337.89,E2 -2337.89} C_VEL
